KUKA KRL program: ps_a_lta_res_x01.src, ps_a_lta_res_x01.dat

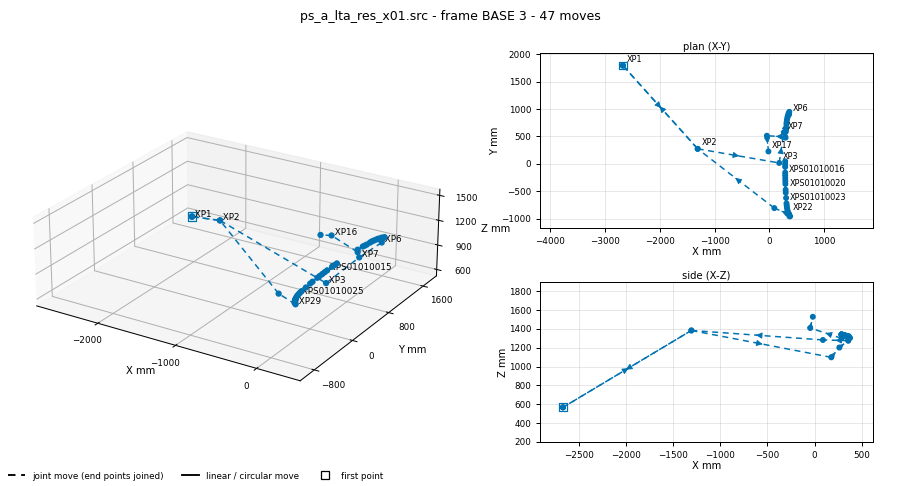
[picture p0: tool path of ps_a_lta_res_x01.src in frame BASE 3, 47 of 49 moves have a stored position in this frame; points joined in program order, loops and branches not executed]
--- ps_a_lta_res_x01.src ---
&ACCESS RVO1
&REL 2
&PARAM DISKPATH = Program/AXOR_ATEGO
DEF ps_a_lta_res_x01( )

;FOLD INI;%{PE}
  ;FOLD BASISTECH INI
    GLOBAL INTERRUPT DECL 3 WHEN $STOPMESS==TRUE DO IR_STOPM ( )
    INTERRUPT ON 3
    BAS (#INITMOV,0 )
  ;ENDFOLD (BASISTECH INI)
;FOLD SPOTTECH INI
USERSPOT(#INIT)
;ENDFOLD (SPOTTECH INI)
;FOLD GRIPPERTECH INI
USER_GRP(0,DUMMY,DUMMY,GDEFAULT)
;ENDFOLD (GRIPPERTECH INI)
  ;FOLD USER INI
    ;Make your modifications here

  ;ENDFOLD (USER INI)
;ENDFOLD (INI)

; Caracterizacao dos meios de producao
; Changes: Solda Respot - ATEGO LTA
; Versao Atual: 07/04/2016
; Ferramenta: GUN X1
; Name: P13.090-R6

chk_w4_wechs_ok ( )     ; CHECK GUN X1

if MaxStandMenge (4) then
  MaxStandmengeErreicht (4)
endif
if Elektrodenwechsel (4) then
 ; e_fraes4 ()
endif

;FOLD PTP P1 Vel=100 % PDAT1 Tool[4]:Gun X1 Base[3]:Atego/Axor;%{PE}%R 8.2.24,%MKUKATPBASIS,%CMOVE,%VPTP,%P 1:PTP, 2:P1, 3:, 5:100, 7:PDAT1
$BWDSTART=FALSE
PDAT_ACT=PPDAT1
FDAT_ACT=FP1
BAS(#PTP_PARAMS,100)
PTP XP1
;ENDFOLD

;FOLD ; Aguarda Liberacao p/ Soldar Respot;%{PE}%R8.3,%MKUKATPBASIS,%CCOMMENT,%VNORMAL,%P 2: Aguarda Liberacao p/ Soldar Respot
;ENDFOLD
;FOLD OUT 3346 'MAGAZINE 3 OCUPADO' State=TRUE ;%{PE}%R 8.2.24,%MKUKATPBASIS,%COUT,%VOUTX,%P 2:3346, 3:MAGAZINE 3 OCUPADO, 5:TRUE, 6:
$OUT[3346]=TRUE
;ENDFOLD
;FOLD WAIT FOR ( IN 3346 'LIB. ROBO SOLDAR RESPOT (ATEGO/AXOR)' );%{PE}%R 8.2.24,%MKUKATPBASIS,%CEXT_WAIT_FOR,%VEXT_WAIT_FOR,%P 2:, 4:, 5:$IN, 6:3346, 7:LIB. ROBO SOLDAR RESPOT (ATEGO/AXOR), 9:
WAIT FOR  ( $IN[3346] )
;ENDFOLD
;FOLD OUT 3346 'MAGAZINE 3 OCUPADO' State=FALSE ;%{PE}%R 8.2.24,%MKUKATPBASIS,%COUT,%VOUTX,%P 2:3346, 3:MAGAZINE 3 OCUPADO, 5:FALSE, 6:
$OUT[3346]=FALSE
;ENDFOLD

;FOLD ; Liga intertravamento  com R4;%{PE}%R8.3,%MKUKATPBASIS,%CCOMMENT,%VNORMAL,%P 2: Liga intertravamento  com R4
;ENDFOLD
;FOLD ; Intertravamento 15 do R4 equivalente ao Intertravamento 15 no R6;%{PE}%R 8.2.24,%MKUKATPBASIS,%CCOMMENT,%VNORMAL,%P 2:Intertravamento 15 do R4 equivalente ao Intertravamento 15 no R6
;ENDFOLD
;FOLD Collision.Monitoring_15_On ;%{PE}%MKUKATPUSER

COLLSTOP( 15, 1 ) ;not Interrupt-Controlled

;ENDFOLD

;FOLD PTP P2 CONT Vel=100 % PDAT2 Tool[4]:Gun X1 Base[3]:Atego/Axor;%{PE}%R 8.2.24,%MKUKATPBASIS,%CMOVE,%VPTP,%P 1:PTP, 2:P2, 3:C_PTP, 5:100, 7:PDAT2
$BWDSTART=FALSE
PDAT_ACT=PPDAT2
FDAT_ACT=FP2
BAS(#PTP_PARAMS,100)
PTP XP2 C_PTP
;ENDFOLD
;FOLD PTP P3 CONT Vel=100 % PDAT3 Tool[4]:Gun X1 Base[3]:Atego/Axor;%{PE}%R 8.2.24,%MKUKATPBASIS,%CMOVE,%VPTP,%P 1:PTP, 2:P3, 3:C_PTP, 5:100, 7:PDAT3
$BWDSTART=FALSE
PDAT_ACT=PPDAT3
FDAT_ACT=FP3
BAS(#PTP_PARAMS,100)
PTP XP3 C_PTP
;ENDFOLD
;FOLD PTP P7 CONT Vel=100 % PDAT6 Tool[4]:Gun X1 Base[3]:Atego/Axor;%{PE}%R 8.2.24,%MKUKATPBASIS,%CMOVE,%VPTP,%P 1:PTP, 2:P7, 3:C_PTP, 5:100, 7:PDAT6
$BWDSTART=FALSE
PDAT_ACT=PPDAT6
FDAT_ACT=FP7
BAS(#PTP_PARAMS,100)
PTP XP7 C_PTP
;ENDFOLD
;FOLD PTP P6 Vel=100 % PDAT5 Tool[4]:Gun X1 Base[3]:Atego/Axor;%{PE}%R 8.2.24,%MKUKATPBASIS,%CMOVE,%VPTP,%P 1:PTP, 2:P6, 3:, 5:100, 7:PDAT5
$BWDSTART=FALSE
PDAT_ACT=PPDAT5
FDAT_ACT=FP6
BAS(#PTP_PARAMS,100)
PTP XP6
;ENDFOLD

;FOLD ; SWP_60_9640;%{PE}%R8.3,%MKUKATPBASIS,%CCOMMENT,%VNORMAL,%P 2: SWP_60_9640
;ENDFOLD
;FOLD LIN PS01010002 CPDAT6 SPOT Gun=2 RETR CLS PgNo1=182 ACTIVE=1 Tool[4]:Gun X1 Base[3]:Atego/Axor;%{PE}%R 8.2.2,%MKUKATPSPOT,%CSPOT,%VLIN,%P 1:LIN, 2:PS01010002, 3:, 5:2, 7:CPDAT6, 10:2, 12:#FIRST, 14:#CLO, 16:182, 18:1, 20:0, 22:0, 24:1, 25:NORMAL
$BWDSTART=FALSE
LDAT_ACT=LCPDAT6
FDAT_ACT=FPS01010002
BAS(#CP_PARAMS,LCPDAT6.VEL)
S_ACT.GUN=2
S_ACT.PAIR=SDEFAULT.PAIR
S_ACT.RETR=#CLO
S_ACT.CLO_TM=1
S_ACT.PGNO1=182
S_ACT.PGNO2=SDEFAULT.PGNO2
S_ACT.PRESS1=SDEFAULT.PRESS1
S_ACT.PRESS2=SDEFAULT.PRESS2
S_READY=FALSE
LIN XPS01010002
USERSPOT(#SPOT, S_ACT)
WAIT FOR S_READY

;ENDFOLD
;FOLD LIN P9 Vel=2 m/s CPDAT5 Tool[4]:Gun X1 Base[3]:Atego/Axor;%{PE}%R 8.2.24,%MKUKATPBASIS,%CMOVE,%VLIN,%P 1:LIN, 2:P9, 3:, 5:2, 7:CPDAT5
$BWDSTART=FALSE
LDAT_ACT=LCPDAT5
FDAT_ACT=FP9
BAS(#CP_PARAMS,2)
LIN XP9
;ENDFOLD

;FOLD ; SWP_60_9638;%{PE}%R8.3,%MKUKATPBASIS,%CCOMMENT,%VNORMAL,%P 2: SWP_60_9638
;ENDFOLD
;FOLD LIN PS01010003 CPDAT4 SPOT Gun=2 RETR CLS PgNo1=182 ACTIVE=1 Tool[4]:Gun X1 Base[3]:Atego/Axor;%{PE}%R 8.2.2,%MKUKATPSPOT,%CSPOT,%VLIN,%P 1:LIN, 2:PS01010003, 3:, 5:2, 7:CPDAT4, 10:2, 12:#FIRST, 14:#CLO, 16:182, 18:1, 20:0, 22:0, 24:1, 25:NORMAL
$BWDSTART=FALSE
LDAT_ACT=LCPDAT4
FDAT_ACT=FPS01010003
BAS(#CP_PARAMS,LCPDAT4.VEL)
S_ACT.GUN=2
S_ACT.PAIR=SDEFAULT.PAIR
S_ACT.RETR=#CLO
S_ACT.CLO_TM=1
S_ACT.PGNO1=182
S_ACT.PGNO2=SDEFAULT.PGNO2
S_ACT.PRESS1=SDEFAULT.PRESS1
S_ACT.PRESS2=SDEFAULT.PRESS2
S_READY=FALSE
LIN XPS01010003
USERSPOT(#SPOT, S_ACT)
WAIT FOR S_READY

;ENDFOLD

;FOLD LIN P10 Vel=2 m/s CPDAT3 Tool[4]:Gun X1 Base[3]:Atego/Axor;%{PE}%R 8.2.24,%MKUKATPBASIS,%CMOVE,%VLIN,%P 1:LIN, 2:P10, 3:, 5:2, 7:CPDAT3
$BWDSTART=FALSE
LDAT_ACT=LCPDAT3
FDAT_ACT=FP10
BAS(#CP_PARAMS,2)
LIN XP10
;ENDFOLD

;FOLD ; SWP_60_9636;%{PE}%R8.3,%MKUKATPBASIS,%CCOMMENT,%VNORMAL,%P 2: SWP_60_9636
;ENDFOLD
;FOLD LIN PS01010004 CPDAT7 SPOT Gun=2 RETR CLS PgNo1=185 ACTIVE=1 Tool[4]:Gun X1 Base[3]:Atego/Axor;%{PE}%R 8.2.2,%MKUKATPSPOT,%CSPOT,%VLIN,%P 1:LIN, 2:PS01010004, 3:, 5:2, 7:CPDAT7, 10:2, 12:#FIRST, 14:#CLO, 16:185, 18:1, 20:0, 22:0, 24:1, 25:NORMAL
$BWDSTART=FALSE
LDAT_ACT=LCPDAT7
FDAT_ACT=FPS01010004
BAS(#CP_PARAMS,LCPDAT7.VEL)
S_ACT.GUN=2
S_ACT.PAIR=SDEFAULT.PAIR
S_ACT.RETR=#CLO
S_ACT.CLO_TM=1
S_ACT.PGNO1=185
S_ACT.PGNO2=SDEFAULT.PGNO2
S_ACT.PRESS1=SDEFAULT.PRESS1
S_ACT.PRESS2=SDEFAULT.PRESS2
S_READY=FALSE
LIN XPS01010004
USERSPOT(#SPOT, S_ACT)
WAIT FOR S_READY

;ENDFOLD

;FOLD ; SWP_60_9634;%{PE}%R8.3,%MKUKATPBASIS,%CCOMMENT,%VNORMAL,%P 2: SWP_60_9634
;ENDFOLD
;FOLD LIN PS01010005 CPDAT8 SPOT Gun=2 RETR CLS PgNo1=181 ACTIVE=1 Tool[4]:Gun X1 Base[3]:Atego/Axor;%{PE}%R 8.2.2,%MKUKATPSPOT,%CSPOT,%VLIN,%P 1:LIN, 2:PS01010005, 3:, 5:2, 7:CPDAT8, 10:2, 12:#FIRST, 14:#CLO, 16:181, 18:1, 20:0, 22:0, 24:1, 25:NORMAL
$BWDSTART=FALSE
LDAT_ACT=LCPDAT8
FDAT_ACT=FPS01010005
BAS(#CP_PARAMS,LCPDAT8.VEL)
S_ACT.GUN=2
S_ACT.PAIR=SDEFAULT.PAIR
S_ACT.RETR=#CLO
S_ACT.CLO_TM=1
S_ACT.PGNO1=181
S_ACT.PGNO2=SDEFAULT.PGNO2
S_ACT.PRESS1=SDEFAULT.PRESS1
S_ACT.PRESS2=SDEFAULT.PRESS2
S_READY=FALSE
LIN XPS01010005
USERSPOT(#SPOT, S_ACT)
WAIT FOR S_READY

;ENDFOLD

;FOLD ; SWP_60_9632;%{PE}%R8.3,%MKUKATPBASIS,%CCOMMENT,%VNORMAL,%P 2: SWP_60_9632
;ENDFOLD
;FOLD LIN PS01010006 CPDAT9 SPOT Gun=2 RETR CLS PgNo1=181 ACTIVE=1 Tool[4]:Gun X1 Base[3]:Atego/Axor;%{PE}%R 8.2.2,%MKUKATPSPOT,%CSPOT,%VLIN,%P 1:LIN, 2:PS01010006, 3:, 5:2, 7:CPDAT9, 10:2, 12:#FIRST, 14:#CLO, 16:181, 18:1, 20:0, 22:0, 24:1, 25:NORMAL
$BWDSTART=FALSE
LDAT_ACT=LCPDAT9
FDAT_ACT=FPS01010006
BAS(#CP_PARAMS,LCPDAT9.VEL)
S_ACT.GUN=2
S_ACT.PAIR=SDEFAULT.PAIR
S_ACT.RETR=#CLO
S_ACT.CLO_TM=1
S_ACT.PGNO1=181
S_ACT.PGNO2=SDEFAULT.PGNO2
S_ACT.PRESS1=SDEFAULT.PRESS1
S_ACT.PRESS2=SDEFAULT.PRESS2
S_READY=FALSE
LIN XPS01010006
USERSPOT(#SPOT, S_ACT)
WAIT FOR S_READY

;ENDFOLD

;FOLD ; SWP_60_9630;%{PE}%R8.3,%MKUKATPBASIS,%CCOMMENT,%VNORMAL,%P 2: SWP_60_9630
;ENDFOLD
;FOLD LIN PS01010008 CPDAT11 SPOT Gun=2 RETR CLS PgNo1=181 ACTIVE=1 Tool[4]:Gun X1 Base[3]:Atego/Axor;%{PE}%R 8.2.2,%MKUKATPSPOT,%CSPOT,%VLIN,%P 1:LIN, 2:PS01010008, 3:, 5:2, 7:CPDAT11, 10:2, 12:#FIRST, 14:#CLO, 16:181, 18:1, 20:0, 22:0, 24:1, 25:NORMAL
$BWDSTART=FALSE
LDAT_ACT=LCPDAT11
FDAT_ACT=FPS01010008
BAS(#CP_PARAMS,LCPDAT11.VEL)
S_ACT.GUN=2
S_ACT.PAIR=SDEFAULT.PAIR
S_ACT.RETR=#CLO
S_ACT.CLO_TM=1
S_ACT.PGNO1=181
S_ACT.PGNO2=SDEFAULT.PGNO2
S_ACT.PRESS1=SDEFAULT.PRESS1
S_ACT.PRESS2=SDEFAULT.PRESS2
S_READY=FALSE
LIN XPS01010008
USERSPOT(#SPOT, S_ACT)
WAIT FOR S_READY

;ENDFOLD

;FOLD ; SWP_60_9628;%{PE}%R8.3,%MKUKATPBASIS,%CCOMMENT,%VNORMAL,%P 2: SWP_60_9628
;ENDFOLD
;FOLD LIN PS01010009 CPDAT12 SPOT Gun=2 RETR CLS PgNo1=181 ACTIVE=1 Tool[4]:Gun X1 Base[3]:Atego/Axor;%{PE}%R 8.2.2,%MKUKATPSPOT,%CSPOT,%VLIN,%P 1:LIN, 2:PS01010009, 3:, 5:2, 7:CPDAT12, 10:2, 12:#FIRST, 14:#CLO, 16:181, 18:1, 20:0, 22:0, 24:1, 25:NORMAL
$BWDSTART=FALSE
LDAT_ACT=LCPDAT12
FDAT_ACT=FPS01010009
BAS(#CP_PARAMS,LCPDAT12.VEL)
S_ACT.GUN=2
S_ACT.PAIR=SDEFAULT.PAIR
S_ACT.RETR=#CLO
S_ACT.CLO_TM=1
S_ACT.PGNO1=181
S_ACT.PGNO2=SDEFAULT.PGNO2
S_ACT.PRESS1=SDEFAULT.PRESS1
S_ACT.PRESS2=SDEFAULT.PRESS2
S_READY=FALSE
LIN XPS01010009
USERSPOT(#SPOT, S_ACT)
WAIT FOR S_READY

;ENDFOLD

;FOLD LIN P13 CONT Vel=2 m/s CPDAT16 Tool[4]:Gun X1 Base[3]:Atego/Axor;%{PE}%R 8.2.24,%MKUKATPBASIS,%CMOVE,%VLIN,%P 1:LIN, 2:P13, 3:C_DIS, 5:2, 7:CPDAT16
$BWDSTART=FALSE
LDAT_ACT=LCPDAT16
FDAT_ACT=FP13
BAS(#CP_PARAMS,2)
LIN XP13 C_DIS
;ENDFOLD
;FOLD ; SWP_60_9624;%{PE}%R8.3,%MKUKATPBASIS,%CCOMMENT,%VNORMAL,%P 2: SWP_60_9624
;ENDFOLD
;FOLD LIN PS01010010 CPDAT15 SPOT Gun=2 RETR CLS PgNo1=186 ACTIVE=1 Tool[4]:Gun X1 Base[3]:Atego/Axor;%{PE}%R 8.2.2,%MKUKATPSPOT,%CSPOT,%VLIN,%P 1:LIN, 2:PS01010010, 3:, 5:2, 7:CPDAT15, 10:2, 12:#FIRST, 14:#CLO, 16:186, 18:1, 20:0, 22:0, 24:1, 25:NORMAL
$BWDSTART=FALSE
LDAT_ACT=LCPDAT15
FDAT_ACT=FPS01010010
BAS(#CP_PARAMS,LCPDAT15.VEL)
S_ACT.GUN=2
S_ACT.PAIR=SDEFAULT.PAIR
S_ACT.RETR=#CLO
S_ACT.CLO_TM=1
S_ACT.PGNO1=186
S_ACT.PGNO2=SDEFAULT.PGNO2
S_ACT.PRESS1=SDEFAULT.PRESS1
S_ACT.PRESS2=SDEFAULT.PRESS2
S_READY=FALSE
LIN XPS01010010
USERSPOT(#SPOT, S_ACT)
WAIT FOR S_READY

;ENDFOLD

;FOLD ; SWP_60_9622;%{PE}%R8.3,%MKUKATPBASIS,%CCOMMENT,%VNORMAL,%P 2: SWP_60_9622
;ENDFOLD
;FOLD LIN PS01010011 CPDAT17 SPOT Gun=2 RETR CLS PgNo1=181 ACTIVE=1 Tool[4]:Gun X1 Base[3]:Atego/Axor;%{PE}%R 8.2.2,%MKUKATPSPOT,%CSPOT,%VLIN,%P 1:LIN, 2:PS01010011, 3:, 5:2, 7:CPDAT17, 10:2, 12:#FIRST, 14:#CLO, 16:181, 18:1, 20:0, 22:0, 24:1, 25:NORMAL
$BWDSTART=FALSE
LDAT_ACT=LCPDAT17
FDAT_ACT=FPS01010011
BAS(#CP_PARAMS,LCPDAT17.VEL)
S_ACT.GUN=2
S_ACT.PAIR=SDEFAULT.PAIR
S_ACT.RETR=#CLO
S_ACT.CLO_TM=1
S_ACT.PGNO1=181
S_ACT.PGNO2=SDEFAULT.PGNO2
S_ACT.PRESS1=SDEFAULT.PRESS1
S_ACT.PRESS2=SDEFAULT.PRESS2
S_READY=FALSE
LIN XPS01010011
USERSPOT(#SPOT, S_ACT)
WAIT FOR S_READY

;ENDFOLD

;FOLD ; SWP_60_9618;%{PE}%R8.3,%MKUKATPBASIS,%CCOMMENT,%VNORMAL,%P 2: SWP_60_9618
;ENDFOLD
;FOLD LIN PS01010012 CPDAT18 SPOT Gun=2 RETR CLS PgNo1=181 ACTIVE=1 Tool[4]:Gun X1 Base[3]:Atego/Axor;%{PE}%R 8.2.2,%MKUKATPSPOT,%CSPOT,%VLIN,%P 1:LIN, 2:PS01010012, 3:, 5:2, 7:CPDAT18, 10:2, 12:#FIRST, 14:#CLO, 16:181, 18:1, 20:0, 22:0, 24:1, 25:NORMAL
$BWDSTART=FALSE
LDAT_ACT=LCPDAT18
FDAT_ACT=FPS01010012
BAS(#CP_PARAMS,LCPDAT18.VEL)
S_ACT.GUN=2
S_ACT.PAIR=SDEFAULT.PAIR
S_ACT.RETR=#CLO
S_ACT.CLO_TM=1
S_ACT.PGNO1=181
S_ACT.PGNO2=SDEFAULT.PGNO2
S_ACT.PRESS1=SDEFAULT.PRESS1
S_ACT.PRESS2=SDEFAULT.PRESS2
S_READY=FALSE
LIN XPS01010012
USERSPOT(#SPOT, S_ACT)
WAIT FOR S_READY

;ENDFOLD

;FOLD LIN P14 Vel=2 m/s CPDAT19 Tool[4]:Gun X1 Base[3]:Atego/Axor;%{PE}%R 8.2.24,%MKUKATPBASIS,%CMOVE,%VLIN,%P 1:LIN, 2:P14, 3:, 5:2, 7:CPDAT19
$BWDSTART=FALSE
LDAT_ACT=LCPDAT19
FDAT_ACT=FP14
BAS(#CP_PARAMS,2)
LIN XP14
;ENDFOLD
;FOLD PTP P16 Vel=100 % PDAT12 Tool[4]:Gun X1 Base[3]:Atego/Axor;%{PE}%R 8.2.24,%MKUKATPBASIS,%CMOVE,%VPTP,%P 1:PTP, 2:P16, 3:, 5:100, 7:PDAT12
$BWDSTART=FALSE
PDAT_ACT=PPDAT12
FDAT_ACT=FP16
BAS(#PTP_PARAMS,100)
PTP XP16
;ENDFOLD
;FOLD PTP P17 CONT Vel=100 % PDAT13 Tool[4]:Gun X1 Base[3]:Atego/Axor;%{PE}%R 8.2.24,%MKUKATPBASIS,%CMOVE,%VPTP,%P 1:PTP, 2:P17, 3:C_PTP, 5:100, 7:PDAT13
$BWDSTART=FALSE
PDAT_ACT=PPDAT13
FDAT_ACT=FP17
BAS(#PTP_PARAMS,100)
PTP XP17 C_PTP
;ENDFOLD
;FOLD PTP P19 CONT Vel=100 % PDAT14 Tool[5]:Gripper Geo G01 00 Base[0];%{PE}%R 8.2.24,%MKUKATPBASIS,%CMOVE,%VPTP,%P 1:PTP, 2:P19, 3:C_PTP, 5:100, 7:PDAT14
$BWDSTART=FALSE
PDAT_ACT=PPDAT14
FDAT_ACT=FP19
BAS(#PTP_PARAMS,100)
PTP XP19 C_PTP
;ENDFOLD
;FOLD PTP P20 Vel=100 % PDAT15 Tool[5]:Gripper Geo G01 00 Base[0];%{PE}%R 8.2.24,%MKUKATPBASIS,%CMOVE,%VPTP,%P 1:PTP, 2:P20, 3:, 5:100, 7:PDAT15
$BWDSTART=FALSE
PDAT_ACT=PPDAT15
FDAT_ACT=FP20
BAS(#PTP_PARAMS,100)
PTP XP20
;ENDFOLD

;FOLD ; SWP_60_9602;%{PE}%R8.3,%MKUKATPBASIS,%CCOMMENT,%VNORMAL,%P 2: SWP_60_9602
;ENDFOLD
;FOLD LIN PS01010013 CPDAT20 SPOT Gun=2 RETR CLS PgNo1=181 ACTIVE=1 Tool[4]:Gun X1 Base[3]:Atego/Axor;%{PE}%R 8.2.2,%MKUKATPSPOT,%CSPOT,%VLIN,%P 1:LIN, 2:PS01010013, 3:, 5:2, 7:CPDAT20, 10:2, 12:#FIRST, 14:#CLO, 16:181, 18:1, 20:0, 22:0, 24:1, 25:NORMAL
$BWDSTART=FALSE
LDAT_ACT=LCPDAT20
FDAT_ACT=FPS01010013
BAS(#CP_PARAMS,LCPDAT20.VEL)
S_ACT.GUN=2
S_ACT.PAIR=SDEFAULT.PAIR
S_ACT.RETR=#CLO
S_ACT.CLO_TM=1
S_ACT.PGNO1=181
S_ACT.PGNO2=SDEFAULT.PGNO2
S_ACT.PRESS1=SDEFAULT.PRESS1
S_ACT.PRESS2=SDEFAULT.PRESS2
S_READY=FALSE
LIN XPS01010013
USERSPOT(#SPOT, S_ACT)
WAIT FOR S_READY

;ENDFOLD

;FOLD ; SWP_60_9600;%{PE}%R8.3,%MKUKATPBASIS,%CCOMMENT,%VNORMAL,%P 2: SWP_60_9600
;ENDFOLD
;FOLD LIN PS01010007 CPDAT10 SPOT Gun=2 RETR CLS PgNo1=186 ACTIVE=1 Tool[4]:Gun X1 Base[3]:Atego/Axor;%{PE}%R 8.2.2,%MKUKATPSPOT,%CSPOT,%VLIN,%P 1:LIN, 2:PS01010007, 3:, 5:2, 7:CPDAT10, 10:2, 12:#FIRST, 14:#CLO, 16:186, 18:1, 20:0, 22:0, 24:1, 25:NORMAL
$BWDSTART=FALSE
LDAT_ACT=LCPDAT10
FDAT_ACT=FPS01010007
BAS(#CP_PARAMS,LCPDAT10.VEL)
S_ACT.GUN=2
S_ACT.PAIR=SDEFAULT.PAIR
S_ACT.RETR=#CLO
S_ACT.CLO_TM=1
S_ACT.PGNO1=186
S_ACT.PGNO2=SDEFAULT.PGNO2
S_ACT.PRESS1=SDEFAULT.PRESS1
S_ACT.PRESS2=SDEFAULT.PRESS2
S_READY=FALSE
LIN XPS01010007
USERSPOT(#SPOT, S_ACT)
WAIT FOR S_READY

;ENDFOLD

;FOLD ; SWP_60_9601;%{PE}%R8.3,%MKUKATPBASIS,%CCOMMENT,%VNORMAL,%P 2: SWP_60_9601
;ENDFOLD
;FOLD LIN PS01010014 CPDAT21 SPOT Gun=2 RETR CLS PgNo1=181 ACTIVE=1 Tool[4]:Gun X1 Base[3]:Atego/Axor;%{PE}%R 8.2.2,%MKUKATPSPOT,%CSPOT,%VLIN,%P 1:LIN, 2:PS01010014, 3:, 5:2, 7:CPDAT21, 10:2, 12:#FIRST, 14:#CLO, 16:181, 18:1, 20:0, 22:0, 24:1, 25:NORMAL
$BWDSTART=FALSE
LDAT_ACT=LCPDAT21
FDAT_ACT=FPS01010014
BAS(#CP_PARAMS,LCPDAT21.VEL)
S_ACT.GUN=2
S_ACT.PAIR=SDEFAULT.PAIR
S_ACT.RETR=#CLO
S_ACT.CLO_TM=1
S_ACT.PGNO1=181
S_ACT.PGNO2=SDEFAULT.PGNO2
S_ACT.PRESS1=SDEFAULT.PRESS1
S_ACT.PRESS2=SDEFAULT.PRESS2
S_READY=FALSE
LIN XPS01010014
USERSPOT(#SPOT, S_ACT)
WAIT FOR S_READY

;ENDFOLD

;FOLD ; SWP_60_9605;%{PE}%R8.3,%MKUKATPBASIS,%CCOMMENT,%VNORMAL,%P 2: SWP_60_9605
;ENDFOLD
;FOLD LIN PS01010015 CPDAT22 SPOT Gun=2 RETR CLS PgNo1=181 ACTIVE=1 Tool[4]:Gun X1 Base[3]:Atego/Axor;%{PE}%R 8.2.2,%MKUKATPSPOT,%CSPOT,%VLIN,%P 1:LIN, 2:PS01010015, 3:, 5:2, 7:CPDAT22, 10:2, 12:#FIRST, 14:#CLO, 16:181, 18:1, 20:0, 22:0, 24:1, 25:NORMAL
$BWDSTART=FALSE
LDAT_ACT=LCPDAT22
FDAT_ACT=FPS01010015
BAS(#CP_PARAMS,LCPDAT22.VEL)
S_ACT.GUN=2
S_ACT.PAIR=SDEFAULT.PAIR
S_ACT.RETR=#CLO
S_ACT.CLO_TM=1
S_ACT.PGNO1=181
S_ACT.PGNO2=SDEFAULT.PGNO2
S_ACT.PRESS1=SDEFAULT.PRESS1
S_ACT.PRESS2=SDEFAULT.PRESS2
S_READY=FALSE
LIN XPS01010015
USERSPOT(#SPOT, S_ACT)
WAIT FOR S_READY

;ENDFOLD

;FOLD ; SWP_60_9607;%{PE}%R8.3,%MKUKATPBASIS,%CCOMMENT,%VNORMAL,%P 2: SWP_60_9607
;ENDFOLD
;FOLD LIN PS01010016 CPDAT23 SPOT Gun=2 RETR CLS PgNo1=181 ACTIVE=1 Tool[4]:Gun X1 Base[3]:Atego/Axor;%{PE}%R 8.2.2,%MKUKATPSPOT,%CSPOT,%VLIN,%P 1:LIN, 2:PS01010016, 3:, 5:2, 7:CPDAT23, 10:2, 12:#FIRST, 14:#CLO, 16:181, 18:1, 20:0, 22:0, 24:1, 25:NORMAL
$BWDSTART=FALSE
LDAT_ACT=LCPDAT23
FDAT_ACT=FPS01010016
BAS(#CP_PARAMS,LCPDAT23.VEL)
S_ACT.GUN=2
S_ACT.PAIR=SDEFAULT.PAIR
S_ACT.RETR=#CLO
S_ACT.CLO_TM=1
S_ACT.PGNO1=181
S_ACT.PGNO2=SDEFAULT.PGNO2
S_ACT.PRESS1=SDEFAULT.PRESS1
S_ACT.PRESS2=SDEFAULT.PRESS2
S_READY=FALSE
LIN XPS01010016
USERSPOT(#SPOT, S_ACT)
WAIT FOR S_READY

;ENDFOLD

;FOLD ; SWP_60_9609;%{PE}%R8.3,%MKUKATPBASIS,%CCOMMENT,%VNORMAL,%P 2: SWP_60_9609
;ENDFOLD
;FOLD LIN PS01010017 CPDAT24 SPOT Gun=2 RETR CLS PgNo1=181 ACTIVE=1 Tool[4]:Gun X1 Base[3]:Atego/Axor;%{PE}%R 8.2.2,%MKUKATPSPOT,%CSPOT,%VLIN,%P 1:LIN, 2:PS01010017, 3:, 5:2, 7:CPDAT24, 10:2, 12:#FIRST, 14:#CLO, 16:181, 18:1, 20:0, 22:0, 24:1, 25:NORMAL
$BWDSTART=FALSE
LDAT_ACT=LCPDAT24
FDAT_ACT=FPS01010017
BAS(#CP_PARAMS,LCPDAT24.VEL)
S_ACT.GUN=2
S_ACT.PAIR=SDEFAULT.PAIR
S_ACT.RETR=#CLO
S_ACT.CLO_TM=1
S_ACT.PGNO1=181
S_ACT.PGNO2=SDEFAULT.PGNO2
S_ACT.PRESS1=SDEFAULT.PRESS1
S_ACT.PRESS2=SDEFAULT.PRESS2
S_READY=FALSE
LIN XPS01010017
USERSPOT(#SPOT, S_ACT)
WAIT FOR S_READY

;ENDFOLD

;FOLD ; SWP_60_9611;%{PE}%R8.3,%MKUKATPBASIS,%CCOMMENT,%VNORMAL,%P 2: SWP_60_9611
;ENDFOLD
;FOLD LIN PS01010018 CPDAT25 SPOT Gun=2 RETR CLS PgNo1=181 ACTIVE=1 Tool[4]:Gun X1 Base[3]:Atego/Axor;%{PE}%R 8.2.2,%MKUKATPSPOT,%CSPOT,%VLIN,%P 1:LIN, 2:PS01010018, 3:, 5:2, 7:CPDAT25, 10:2, 12:#FIRST, 14:#CLO, 16:181, 18:1, 20:0, 22:0, 24:1, 25:NORMAL
$BWDSTART=FALSE
LDAT_ACT=LCPDAT25
FDAT_ACT=FPS01010018
BAS(#CP_PARAMS,LCPDAT25.VEL)
S_ACT.GUN=2
S_ACT.PAIR=SDEFAULT.PAIR
S_ACT.RETR=#CLO
S_ACT.CLO_TM=1
S_ACT.PGNO1=181
S_ACT.PGNO2=SDEFAULT.PGNO2
S_ACT.PRESS1=SDEFAULT.PRESS1
S_ACT.PRESS2=SDEFAULT.PRESS2
S_READY=FALSE
LIN XPS01010018
USERSPOT(#SPOT, S_ACT)
WAIT FOR S_READY

;ENDFOLD

;FOLD ; SWP_60_9613;%{PE}%R8.3,%MKUKATPBASIS,%CCOMMENT,%VNORMAL,%P 2: SWP_60_9613
;ENDFOLD
;FOLD LIN PS01010019 CPDAT26 SPOT Gun=2 RETR CLS PgNo1=181 ACTIVE=1 Tool[4]:Gun X1 Base[3]:Atego/Axor;%{PE}%R 8.2.2,%MKUKATPSPOT,%CSPOT,%VLIN,%P 1:LIN, 2:PS01010019, 3:, 5:2, 7:CPDAT26, 10:2, 12:#FIRST, 14:#CLO, 16:181, 18:1, 20:0, 22:0, 24:1, 25:NORMAL
$BWDSTART=FALSE
LDAT_ACT=LCPDAT26
FDAT_ACT=FPS01010019
BAS(#CP_PARAMS,LCPDAT26.VEL)
S_ACT.GUN=2
S_ACT.PAIR=SDEFAULT.PAIR
S_ACT.RETR=#CLO
S_ACT.CLO_TM=1
S_ACT.PGNO1=181
S_ACT.PGNO2=SDEFAULT.PGNO2
S_ACT.PRESS1=SDEFAULT.PRESS1
S_ACT.PRESS2=SDEFAULT.PRESS2
S_READY=FALSE
LIN XPS01010019
USERSPOT(#SPOT, S_ACT)
WAIT FOR S_READY

;ENDFOLD

;FOLD ; SWP_60_9617;%{PE}%R8.3,%MKUKATPBASIS,%CCOMMENT,%VNORMAL,%P 2: SWP_60_9617
;ENDFOLD
;FOLD LIN PS01010020 CPDAT27 SPOT Gun=2 RETR CLS PgNo1=181 ACTIVE=1 Tool[4]:Gun X1 Base[3]:Atego/Axor;%{PE}%R 8.2.2,%MKUKATPSPOT,%CSPOT,%VLIN,%P 1:LIN, 2:PS01010020, 3:, 5:2, 7:CPDAT27, 10:2, 12:#FIRST, 14:#CLO, 16:181, 18:1, 20:0, 22:0, 24:1, 25:NORMAL
$BWDSTART=FALSE
LDAT_ACT=LCPDAT27
FDAT_ACT=FPS01010020
BAS(#CP_PARAMS,LCPDAT27.VEL)
S_ACT.GUN=2
S_ACT.PAIR=SDEFAULT.PAIR
S_ACT.RETR=#CLO
S_ACT.CLO_TM=1
S_ACT.PGNO1=181
S_ACT.PGNO2=SDEFAULT.PGNO2
S_ACT.PRESS1=SDEFAULT.PRESS1
S_ACT.PRESS2=SDEFAULT.PRESS2
S_READY=FALSE
LIN XPS01010020
USERSPOT(#SPOT, S_ACT)
WAIT FOR S_READY

;ENDFOLD

;FOLD ; SWP_60_9619;%{PE}%R8.3,%MKUKATPBASIS,%CCOMMENT,%VNORMAL,%P 2: SWP_60_9619
;ENDFOLD
;FOLD LIN PS01010021 CPDAT28 SPOT Gun=2 RETR CLS PgNo1=181 ACTIVE=1 Tool[4]:Gun X1 Base[3]:Atego/Axor;%{PE}%R 8.2.2,%MKUKATPSPOT,%CSPOT,%VLIN,%P 1:LIN, 2:PS01010021, 3:, 5:2, 7:CPDAT28, 10:2, 12:#FIRST, 14:#CLO, 16:181, 18:1, 20:0, 22:0, 24:1, 25:NORMAL
$BWDSTART=FALSE
LDAT_ACT=LCPDAT28
FDAT_ACT=FPS01010021
BAS(#CP_PARAMS,LCPDAT28.VEL)
S_ACT.GUN=2
S_ACT.PAIR=SDEFAULT.PAIR
S_ACT.RETR=#CLO
S_ACT.CLO_TM=1
S_ACT.PGNO1=181
S_ACT.PGNO2=SDEFAULT.PGNO2
S_ACT.PRESS1=SDEFAULT.PRESS1
S_ACT.PRESS2=SDEFAULT.PRESS2
S_READY=FALSE
LIN XPS01010021
USERSPOT(#SPOT, S_ACT)
WAIT FOR S_READY

;ENDFOLD

;FOLD ; SWP_60_9623;%{PE}%R8.3,%MKUKATPBASIS,%CCOMMENT,%VNORMAL,%P 2: SWP_60_9623
;ENDFOLD
;FOLD LIN PS01010022 CPDAT29 SPOT Gun=2 RETR CLS PgNo1=186 ACTIVE=1 Tool[4]:Gun X1 Base[3]:Atego/Axor;%{PE}%R 8.2.2,%MKUKATPSPOT,%CSPOT,%VLIN,%P 1:LIN, 2:PS01010022, 3:, 5:2, 7:CPDAT29, 10:2, 12:#FIRST, 14:#CLO, 16:186, 18:1, 20:0, 22:0, 24:1, 25:NORMAL
$BWDSTART=FALSE
LDAT_ACT=LCPDAT29
FDAT_ACT=FPS01010022
BAS(#CP_PARAMS,LCPDAT29.VEL)
S_ACT.GUN=2
S_ACT.PAIR=SDEFAULT.PAIR
S_ACT.RETR=#CLO
S_ACT.CLO_TM=1
S_ACT.PGNO1=186
S_ACT.PGNO2=SDEFAULT.PGNO2
S_ACT.PRESS1=SDEFAULT.PRESS1
S_ACT.PRESS2=SDEFAULT.PRESS2
S_READY=FALSE
LIN XPS01010022
USERSPOT(#SPOT, S_ACT)
WAIT FOR S_READY

;ENDFOLD

;FOLD ; SWP_60_9627(old 9625);%{PE}%R8.3,%MKUKATPBASIS,%CCOMMENT,%VNORMAL,%P 2: SWP_60_9627(old 9625)
;ENDFOLD
;FOLD LIN PS01010023 CPDAT30 SPOT Gun=2 RETR CLS PgNo1=186 ACTIVE=1 Tool[4]:Gun X1 Base[3]:Atego/Axor;%{PE}%R 8.2.2,%MKUKATPSPOT,%CSPOT,%VLIN,%P 1:LIN, 2:PS01010023, 3:, 5:2, 7:CPDAT30, 10:2, 12:#FIRST, 14:#CLO, 16:186, 18:1, 20:0, 22:0, 24:1, 25:NORMAL
$BWDSTART=FALSE
LDAT_ACT=LCPDAT30
FDAT_ACT=FPS01010023
BAS(#CP_PARAMS,LCPDAT30.VEL)
S_ACT.GUN=2
S_ACT.PAIR=SDEFAULT.PAIR
S_ACT.RETR=#CLO
S_ACT.CLO_TM=1
S_ACT.PGNO1=186
S_ACT.PGNO2=SDEFAULT.PGNO2
S_ACT.PRESS1=SDEFAULT.PRESS1
S_ACT.PRESS2=SDEFAULT.PRESS2
S_READY=FALSE
LIN XPS01010023
USERSPOT(#SPOT, S_ACT)
WAIT FOR S_READY

;ENDFOLD

;FOLD ; Desliga intertravamento  com R4;%{PE}%R8.3,%MKUKATPBASIS,%CCOMMENT,%VNORMAL,%P 2: Desliga intertravamento  com R4
;ENDFOLD
;FOLD ; Intertravamento 15 do R4 equivalente ao Intertravamento 15 no R6;%{PE}%R 8.2.24,%MKUKATPBASIS,%CCOMMENT,%VNORMAL,%P 2:Intertravamento 15 do R4 equivalente ao Intertravamento 15 no R6
;ENDFOLD
;FOLD Collision.Monitoring_15_Off . ;%{PE}%MKUKATPUSER

COLLSTOP( 15, 2+0 )

;ENDFOLD

;FOLD ; SWP_60_9629;%{PE}%R8.3,%MKUKATPBASIS,%CCOMMENT,%VNORMAL,%P 2: SWP_60_9629
;ENDFOLD
;FOLD LIN PS01010024 CPDAT31 SPOT Gun=2 RETR CLS PgNo1=181 ACTIVE=1 Tool[4]:Gun X1 Base[3]:Atego/Axor;%{PE}%R 8.2.2,%MKUKATPSPOT,%CSPOT,%VLIN,%P 1:LIN, 2:PS01010024, 3:, 5:2, 7:CPDAT31, 10:2, 12:#FIRST, 14:#CLO, 16:181, 18:1, 20:0, 22:0, 24:1, 25:NORMAL
$BWDSTART=FALSE
LDAT_ACT=LCPDAT31
FDAT_ACT=FPS01010024
BAS(#CP_PARAMS,LCPDAT31.VEL)
S_ACT.GUN=2
S_ACT.PAIR=SDEFAULT.PAIR
S_ACT.RETR=#CLO
S_ACT.CLO_TM=1
S_ACT.PGNO1=181
S_ACT.PGNO2=SDEFAULT.PGNO2
S_ACT.PRESS1=SDEFAULT.PRESS1
S_ACT.PRESS2=SDEFAULT.PRESS2
S_READY=FALSE
LIN XPS01010024
USERSPOT(#SPOT, S_ACT)
WAIT FOR S_READY

;ENDFOLD

;FOLD ; SWP_60_9631;%{PE}%R8.3,%MKUKATPBASIS,%CCOMMENT,%VNORMAL,%P 2: SWP_60_9631
;ENDFOLD
;FOLD LIN PS01010025 CPDAT32 SPOT Gun=2 RETR CLS PgNo1=181 ACTIVE=1 Tool[4]:Gun X1 Base[3]:Atego/Axor;%{PE}%R 8.2.2,%MKUKATPSPOT,%CSPOT,%VLIN,%P 1:LIN, 2:PS01010025, 3:, 5:2, 7:CPDAT32, 10:2, 12:#FIRST, 14:#CLO, 16:181, 18:1, 20:0, 22:0, 24:1, 25:NORMAL
$BWDSTART=FALSE
LDAT_ACT=LCPDAT32
FDAT_ACT=FPS01010025
BAS(#CP_PARAMS,LCPDAT32.VEL)
S_ACT.GUN=2
S_ACT.PAIR=SDEFAULT.PAIR
S_ACT.RETR=#CLO
S_ACT.CLO_TM=1
S_ACT.PGNO1=181
S_ACT.PGNO2=SDEFAULT.PGNO2
S_ACT.PRESS1=SDEFAULT.PRESS1
S_ACT.PRESS2=SDEFAULT.PRESS2
S_READY=FALSE
LIN XPS01010025
USERSPOT(#SPOT, S_ACT)
WAIT FOR S_READY

;ENDFOLD

;FOLD ; SWP_60_9633;%{PE}%R8.3,%MKUKATPBASIS,%CCOMMENT,%VNORMAL,%P 2: SWP_60_9633
;ENDFOLD
;FOLD LIN PS01010026 CPDAT33 SPOT Gun=2 RETR CLS PgNo1=181 ACTIVE=1 Tool[4]:Gun X1 Base[3]:Atego/Axor;%{PE}%R 8.2.2,%MKUKATPSPOT,%CSPOT,%VLIN,%P 1:LIN, 2:PS01010026, 3:, 5:2, 7:CPDAT33, 10:2, 12:#FIRST, 14:#CLO, 16:181, 18:1, 20:0, 22:0, 24:1, 25:NORMAL
$BWDSTART=FALSE
LDAT_ACT=LCPDAT33
FDAT_ACT=FPS01010026
BAS(#CP_PARAMS,LCPDAT33.VEL)
S_ACT.GUN=2
S_ACT.PAIR=SDEFAULT.PAIR
S_ACT.RETR=#CLO
S_ACT.CLO_TM=1
S_ACT.PGNO1=181
S_ACT.PGNO2=SDEFAULT.PGNO2
S_ACT.PRESS1=SDEFAULT.PRESS1
S_ACT.PRESS2=SDEFAULT.PRESS2
S_READY=FALSE
LIN XPS01010026
USERSPOT(#SPOT, S_ACT)
WAIT FOR S_READY

;ENDFOLD

;FOLD ; SWP_60_9635;%{PE}%R8.3,%MKUKATPBASIS,%CCOMMENT,%VNORMAL,%P 2: SWP_60_9635
;ENDFOLD
;FOLD LIN PS01010027 CPDAT34 SPOT Gun=2 RETR CLS PgNo1=185 ACTIVE=1 Tool[4]:Gun X1 Base[3]:Atego/Axor;%{PE}%R 8.2.2,%MKUKATPSPOT,%CSPOT,%VLIN,%P 1:LIN, 2:PS01010027, 3:, 5:2, 7:CPDAT34, 10:2, 12:#FIRST, 14:#CLO, 16:185, 18:1, 20:0, 22:0, 24:1, 25:NORMAL
$BWDSTART=FALSE
LDAT_ACT=LCPDAT34
FDAT_ACT=FPS01010027
BAS(#CP_PARAMS,LCPDAT34.VEL)
S_ACT.GUN=2
S_ACT.PAIR=SDEFAULT.PAIR
S_ACT.RETR=#CLO
S_ACT.CLO_TM=1
S_ACT.PGNO1=185
S_ACT.PGNO2=SDEFAULT.PGNO2
S_ACT.PRESS1=SDEFAULT.PRESS1
S_ACT.PRESS2=SDEFAULT.PRESS2
S_READY=FALSE
LIN XPS01010027
USERSPOT(#SPOT, S_ACT)
WAIT FOR S_READY

;ENDFOLD

;FOLD LIN P22 Vel=2 m/s CPDAT35 Tool[4]:Gun X1 Base[3]:Atego/Axor;%{PE}%R 8.2.24,%MKUKATPBASIS,%CMOVE,%VLIN,%P 1:LIN, 2:P22, 3:, 5:2, 7:CPDAT35
$BWDSTART=FALSE
LDAT_ACT=LCPDAT35
FDAT_ACT=FP22
BAS(#CP_PARAMS,2)
LIN XP22
;ENDFOLD

;FOLD ; SWP_60_9637;%{PE}%R8.3,%MKUKATPBASIS,%CCOMMENT,%VNORMAL,%P 2: SWP_60_9637
;ENDFOLD
;FOLD LIN PS01010028 CPDAT36 SPOT Gun=2 RETR CLS PgNo1=184 ACTIVE=1 Tool[4]:Gun X1 Base[3]:Atego/Axor;%{PE}%R 8.2.2,%MKUKATPSPOT,%CSPOT,%VLIN,%P 1:LIN, 2:PS01010028, 3:, 5:2, 7:CPDAT36, 10:2, 12:#FIRST, 14:#CLO, 16:184, 18:1, 20:0, 22:0, 24:1, 25:NORMAL
$BWDSTART=FALSE
LDAT_ACT=LCPDAT36
FDAT_ACT=FPS01010028
BAS(#CP_PARAMS,LCPDAT36.VEL)
S_ACT.GUN=2
S_ACT.PAIR=SDEFAULT.PAIR
S_ACT.RETR=#CLO
S_ACT.CLO_TM=1
S_ACT.PGNO1=184
S_ACT.PGNO2=SDEFAULT.PGNO2
S_ACT.PRESS1=SDEFAULT.PRESS1
S_ACT.PRESS2=SDEFAULT.PRESS2
S_READY=FALSE
LIN XPS01010028
USERSPOT(#SPOT, S_ACT)
WAIT FOR S_READY

;ENDFOLD

;FOLD LIN P23 Vel=2 m/s CPDAT37 Tool[4]:Gun X1 Base[3]:Atego/Axor;%{PE}%R 8.2.24,%MKUKATPBASIS,%CMOVE,%VLIN,%P 1:LIN, 2:P23, 3:, 5:2, 7:CPDAT37
$BWDSTART=FALSE
LDAT_ACT=LCPDAT37
FDAT_ACT=FP23
BAS(#CP_PARAMS,2)
LIN XP23
;ENDFOLD
;FOLD LIN P24 Vel=2 m/s CPDAT38 Tool[4]:Gun X1 Base[3]:Atego/Axor;%{PE}%R 8.2.24,%MKUKATPBASIS,%CMOVE,%VLIN,%P 1:LIN, 2:P24, 3:, 5:2, 7:CPDAT38
$BWDSTART=FALSE
LDAT_ACT=LCPDAT38
FDAT_ACT=FP24
BAS(#CP_PARAMS,2)
LIN XP24
;ENDFOLD

;FOLD ; Liga intertravamento  com R4;%{PE}%R8.3,%MKUKATPBASIS,%CCOMMENT,%VNORMAL,%P 2: Liga intertravamento  com R4
;ENDFOLD
;FOLD ; Intertravamento 15 do R4 equivalente ao Intertravamento 15 no R6;%{PE}%R 8.2.24,%MKUKATPBASIS,%CCOMMENT,%VNORMAL,%P 2:Intertravamento 15 do R4 equivalente ao Intertravamento 15 no R6
;ENDFOLD
;FOLD Collision.Monitoring_15_On ;%{PE}%MKUKATPUSER

COLLSTOP( 15, 1 ) ;not Interrupt-Controlled

;ENDFOLD

;FOLD ; SWP_60_9639;%{PE}%R8.3,%MKUKATPBASIS,%CCOMMENT,%VNORMAL,%P 2: SWP_60_9639
;ENDFOLD
;FOLD LIN PS01010029 CPDAT40 SPOT Gun=2 RETR OPN PgNo1=184 ACTIVE=1 Tool[4]:Gun X1 Base[3]:Atego/Axor;%{PE}%R 8.2.2,%MKUKATPSPOT,%CSPOT,%VLIN,%P 1:LIN, 2:PS01010029, 3:, 5:2, 7:CPDAT40, 10:2, 12:#FIRST, 14:#OPN, 16:184, 18:1, 20:0, 22:0, 24:1, 25:NORMAL
$BWDSTART=FALSE
LDAT_ACT=LCPDAT40
FDAT_ACT=FPS01010029
BAS(#CP_PARAMS,LCPDAT40.VEL)
S_ACT.GUN=2
S_ACT.PAIR=SDEFAULT.PAIR
S_ACT.RETR=#OPN
S_ACT.CLO_TM=1
S_ACT.PGNO1=184
S_ACT.PGNO2=SDEFAULT.PGNO2
S_ACT.PRESS1=SDEFAULT.PRESS1
S_ACT.PRESS2=SDEFAULT.PRESS2
S_READY=FALSE
LIN XPS01010029
USERSPOT(#SPOT, S_ACT)
WAIT FOR S_READY

;ENDFOLD

;FOLD LIN P29 Vel=2 m/s CPDAT41 Tool[4]:Gun X1 Base[3]:Atego/Axor;%{PE}%R 8.2.24,%MKUKATPBASIS,%CMOVE,%VLIN,%P 1:LIN, 2:P29, 3:, 5:2, 7:CPDAT41
$BWDSTART=FALSE
LDAT_ACT=LCPDAT41
FDAT_ACT=FP29
BAS(#CP_PARAMS,2)
LIN XP29
;ENDFOLD
;FOLD PTP P30 CONT Vel=100 % PDAT19 Tool[4]:Gun X1 Base[3]:Atego/Axor;%{PE}%R 8.2.24,%MKUKATPBASIS,%CMOVE,%VPTP,%P 1:PTP, 2:P30, 3:C_PTP, 5:100, 7:PDAT19
$BWDSTART=FALSE
PDAT_ACT=PPDAT19
FDAT_ACT=FP30
BAS(#PTP_PARAMS,100)
PTP XP30 C_PTP
;ENDFOLD
;FOLD PTP P31 CONT Vel=100 % PDAT20 Tool[4]:Gun X1 Base[3]:Atego/Axor;%{PE}%R 8.2.24,%MKUKATPBASIS,%CMOVE,%VPTP,%P 1:PTP, 2:P31, 3:C_PTP, 5:100, 7:PDAT20
$BWDSTART=FALSE
PDAT_ACT=PPDAT20
FDAT_ACT=FP31
BAS(#PTP_PARAMS,100)
PTP XP31 C_PTP
;ENDFOLD
;FOLD PTP P32 Vel=100 % PDAT21 Tool[4]:Gun X1 Base[3]:Atego/Axor;%{PE}%R 8.2.24,%MKUKATPBASIS,%CMOVE,%VPTP,%P 1:PTP, 2:P32, 3:, 5:100, 7:PDAT21
$BWDSTART=FALSE
PDAT_ACT=PPDAT21
FDAT_ACT=FP32
BAS(#PTP_PARAMS,100)
PTP XP32
;ENDFOLD

;FOLD ; Desliga intertravamento  com R4;%{PE}%R8.3,%MKUKATPBASIS,%CCOMMENT,%VNORMAL,%P 2: Desliga intertravamento  com R4
;ENDFOLD
;FOLD ; Intertravamento 15 do R4 equivalente ao Intertravamento 15 no R6;%{PE}%R 8.2.24,%MKUKATPBASIS,%CCOMMENT,%VNORMAL,%P 2:Intertravamento 15 do R4 equivalente ao Intertravamento 15 no R6
;ENDFOLD
;FOLD Collision.Monitoring_15_Off . ;%{PE}%MKUKATPUSER

COLLSTOP( 15, 2+0 )

;ENDFOLD

;FOLD ; Libera Dispositivo;%{PE}%R8.3,%MKUKATPBASIS,%CCOMMENT,%VNORMAL,%P 2: Libera Dispositivo
;ENDFOLD
;FOLD OUT 3346 'MAGAZINE 3 OCUPADO' State=TRUE CONT;%{PE}%R 8.2.24,%MKUKATPBASIS,%COUT,%VOUTX,%P 2:3346, 3:MAGAZINE 3 OCUPADO, 5:TRUE, 6:CONTINUE
CONTINUE
$OUT[3346]=TRUE
;ENDFOLD

if FraesAnf (4) then
f_fraes4 ()
endif

;FOLD PTP P33 Vel=100 % PDAT22 Tool[4]:Gun X1 Base[3]:Atego/Axor;%{PE}%R 8.2.24,%MKUKATPBASIS,%CMOVE,%VPTP,%P 1:PTP, 2:P33, 3:, 5:100, 7:PDAT22
$BWDSTART=FALSE
PDAT_ACT=PPDAT22
FDAT_ACT=FP33
BAS(#PTP_PARAMS,100)
PTP XP33
;ENDFOLD
END

--- ps_a_lta_res_x01.dat ---
&ACCESS RVO1
&REL 2
&PARAM DISKPATH = Program/AXOR_ATEGO
DEFDAT ps_a_lta_res_x01
;FOLD EXTERNAL DECLARATIONS;%{PE}%MKUKATPBASIS,%CEXT,%VCOMMON,%P
;FOLD BASISTECH EXT;%{PE}%MKUKATPBASIS,%CEXT,%VEXT,%P
EXT  BAS (BAS_COMMAND  :IN,REAL  :IN )
DECL INT SUCCESS
;ENDFOLD (BASISTECH EXT)
;FOLD USER EXT;%{E}%MKUKATPUSER,%CEXT,%VEXT,%P
;Make your modifications here
;ENDFOLD (USER EXT)
;ENDFOLD (EXTERNAL DECLARATIONS)

;# ============ START PATH : ps_a_lta_res_x01 =============
DECL FDAT Fxp8={TOOL_NO 4,BASE_NO 3,IPO_FRAME #BASE,POINT2[] " "}
DECL PDAT PP_OLP1={VEL 100.0,ACC 100.0,APO_DIST 0.0}
DECL E6POS Xxp8={X -2671.84912,Y 1793.97302,Z 566.737,A -2.42820001,B 58.0560989,C 1.01139998,S 2,T 3}
DECL FDAT Fxp10={TOOL_NO 4,BASE_NO 3,IPO_FRAME #BASE,POINT2[] " "}
DECL PDAT PP_OLP2={VEL 100.0,ACC 100.0,APO_DIST 0.0}
DECL E6POS Xxp10={X -1308.078,Y 274.528015,Z 1383.49097,A -11.6739998,B 10.1196003,C -74.1667023,S 2,T 11}
DECL FDAT Fxp20={TOOL_NO 4,BASE_NO 3,IPO_FRAME #BASE,POINT2[] " "}
DECL PDAT PP_OLP3={VEL 100.0,ACC 50.0,APO_DIST 0.0}
DECL E6POS Xxp20={X 178.113007,Y 17.2910004,Z 1098.07605,A 11.9650002,B 9.40390015,C -82.9534988,S 2,T 11}
DECL FDAT Fx1005={TOOL_NO 4,BASE_NO 3,IPO_FRAME #BASE,POINT2[] " "}
DECL E6POS Xx1005={X 338.674988,Y 935.075989,Z 1286.09204,A 34.7946014,B -38.0540009,C -65.3376999,S 2,T 11}
DECL LDAT LL_OLP1={VEL 2.0,ACC 100.0,APO_DIST 1.0,APO_FAC 0.0,ORI_TYP #VAR,CIRC_TYP #BASE,JERK_FAC 50.0}
DECL FDAT Fx1010={TOOL_NO 4,BASE_NO 3,IPO_FRAME #BASE,POINT2[] " "}
DECL E6POS Xx1010={X 371.002014,Y 957.528015,Z 1316.90698,A 34.7947006,B -38.0540009,C -65.3376007,S 2,T 11}
DECL LDAT LL_OLP2={VEL 2.0,ACC 100.0,APO_DIST 1.0,APO_FAC 0.0,ORI_TYP #VAR,CIRC_TYP #BASE,JERK_FAC 50.0}
DECL FDAT Fxswp_6={TOOL_NO 4,BASE_NO 3,IPO_FRAME #BASE,POINT2[] " "}
DECL SPOT_TYPE SS_OLP1={GUN 2,PAIR #FIRST,RETR #CLO,CLO_TM 1,PGNO1 182,PRESS1 0.0,PGNO2 0,PRESS2 0.0}
DECL E6POS Xxswp_6={X 361.389008,Y 946.713989,Z 1327.31006,A 34.7943993,B -38.0540009,C -65.3374023,S 2,T 11}
DECL LDAT LL_OLP3={VEL 2.0,ACC 100.0,APO_DIST 0.0,APO_FAC 0.0,ORI_TYP #VAR,CIRC_TYP #BASE,JERK_FAC 50.0}
DECL FDAT Fx1015={TOOL_NO 4,BASE_NO 3,IPO_FRAME #BASE,POINT2[] " "}
DECL E6POS Xx1015={X 371.001007,Y 957.525024,Z 1316.90601,A 34.7947006,B -38.0540009,C -65.3376999,S 2,T 11}
DECL LDAT LL_OLP4={VEL 2.0,ACC 100.0,APO_DIST 1.0,APO_FAC 0.0,ORI_TYP #VAR,CIRC_TYP #BASE,JERK_FAC 50.0}
DECL FDAT Fxswp_6_1={TOOL_NO 4,BASE_NO 3,IPO_FRAME #BASE,POINT2[] " "}
DECL SPOT_TYPE SS_OLP2={GUN 2,PAIR #FIRST,RETR #CLO,CLO_TM 1,PGNO1 182,PRESS1 0.0,PGNO2 0,PRESS2 0.0}
DECL E6POS Xxswp_6_1={X 344.567993,Y 912.476013,Z 1332.31006,A 51.0245018,B -39.1311989,C -64.2306976,S 2,T 11}
DECL LDAT LL_OLP5={VEL 2.0,ACC 100.0,APO_DIST 0.0,APO_FAC 0.0,ORI_TYP #VAR,CIRC_TYP #BASE,JERK_FAC 50.0}
DECL FDAT Fx1030={TOOL_NO 4,BASE_NO 3,IPO_FRAME #BASE,POINT2[] " "}
DECL E6POS Xx1030={X 344.359985,Y 891.754028,Z 1333.81995,A 56.9338989,B -41.1417999,C -62.901001,S 2,T 11}
DECL LDAT LL_OLP6={VEL 2.0,ACC 100.0,APO_DIST 1.0,APO_FAC 0.0,ORI_TYP #VAR,CIRC_TYP #BASE,JERK_FAC 50.0}
DECL FDAT Fxswp_6_2={TOOL_NO 4,BASE_NO 3,IPO_FRAME #BASE,POINT2[] " "}
DECL SPOT_TYPE SS_OLP3={GUN 2,PAIR #FIRST,RETR #CLO,CLO_TM 1,PGNO1 185,PRESS1 0.0,PGNO2 0,PRESS2 0.0}
DECL E6POS Xxswp_6_2={X 331.682007,Y 863.525024,Z 1333.83398,A 56.9338989,B -41.1417999,C -62.901001,S 2,T 11}
DECL LDAT LL_OLP7={VEL 2.0,ACC 100.0,APO_DIST 0.0,APO_FAC 0.0,ORI_TYP #VAR,CIRC_TYP #BASE,JERK_FAC 50.0}
DECL FDAT Fxswp_6_3={TOOL_NO 4,BASE_NO 3,IPO_FRAME #BASE,POINT2[] " "}
DECL SPOT_TYPE SS_OLP4={GUN 2,PAIR #FIRST,RETR #CLO,CLO_TM 1,PGNO1 181,PRESS1 0.0,PGNO2 0,PRESS2 0.0}
DECL E6POS Xxswp_6_3={X 324.64801,Y 835.888977,Z 1335.92297,A 64.0038986,B -37.8157997,C -65.0102997,S 2,T 11}
DECL LDAT LL_OLP8={VEL 2.0,ACC 100.0,APO_DIST 0.0,APO_FAC 0.0,ORI_TYP #VAR,CIRC_TYP #BASE,JERK_FAC 50.0}
DECL FDAT Fxswp_6_4={TOOL_NO 4,BASE_NO 3,IPO_FRAME #BASE,POINT2[] " "}
DECL SPOT_TYPE SS_OLP5={GUN 2,PAIR #FIRST,RETR #CLO,CLO_TM 1,PGNO1 181,PRESS1 0.0,PGNO2 0,PRESS2 0.0}
DECL E6POS Xxswp_6_4={X 318.389008,Y 798.062012,Z 1336.797,A 63.0040016,B -41.4422989,C -63.5331001,S 2,T 11}
DECL LDAT LL_OLP9={VEL 2.0,ACC 100.0,APO_DIST 0.0,APO_FAC 0.0,ORI_TYP #VAR,CIRC_TYP #BASE,JERK_FAC 50.0}
DECL FDAT Fxswp_6_5={TOOL_NO 4,BASE_NO 3,IPO_FRAME #BASE,POINT2[] " "}
DECL SPOT_TYPE SS_OLP6={GUN 2,PAIR #FIRST,RETR #CLO,CLO_TM 1,PGNO1 181,PRESS1 0.0,PGNO2 0,PRESS2 0.0}
DECL E6POS Xxswp_6_5={X 313.28299,Y 758.213989,Z 1338.11304,A 65.8960037,B -39.6694984,C -64.0615997,S 2,T 11}
DECL LDAT LL_OLP10={VEL 2.0,ACC 100.0,APO_DIST 0.0,APO_FAC 0.0,ORI_TYP #VAR,CIRC_TYP #BASE,JERK_FAC 50.0}
DECL FDAT Fxswp_6_6={TOOL_NO 4,BASE_NO 3,IPO_FRAME #BASE,POINT2[] " "}
DECL SPOT_TYPE SS_OLP7={GUN 2,PAIR #FIRST,RETR #CLO,CLO_TM 1,PGNO1 181,PRESS1 0.0,PGNO2 0,PRESS2 0.0}
DECL E6POS Xxswp_6_6={X 309.087006,Y 718.695007,Z 1339.03503,A 69.3459015,B -38.6236992,C -68.3812027,S 2,T 11}
DECL LDAT LL_OLP11={VEL 2.0,ACC 100.0,APO_DIST 0.0,APO_FAC 0.0,ORI_TYP #VAR,CIRC_TYP #BASE,JERK_FAC 50.0}
DECL FDAT Fx1035={TOOL_NO 4,BASE_NO 3,IPO_FRAME #BASE,POINT2[] " "}
DECL E6POS Xx1035={X 297.544006,Y 716.080017,Z 1298.703,A 69.3459015,B -38.6237984,C -68.3811035,S 2,T 11}
DECL LDAT LL_OLP12={VEL 2.0,ACC 100.0,APO_DIST 1.0,APO_FAC 0.0,ORI_TYP #VAR,CIRC_TYP #BASE,JERK_FAC 50.0}
DECL FDAT Fx1040={TOOL_NO 4,BASE_NO 3,IPO_FRAME #BASE,POINT2[] " "}
DECL PDAT PP_OLP4={VEL 100.0,ACC 100.0,APO_DIST 0.0}
DECL E6POS Xx1040={X 290.720001,Y 611.52002,Z 1294.58899,A 70.504303,B -35.8750992,C -65.2176971,S 2,T 11}
DECL FDAT Fxswp_6_7={TOOL_NO 4,BASE_NO 3,IPO_FRAME #BASE,POINT2[] " "}
DECL SPOT_TYPE SS_OLP8={GUN 2,PAIR #FIRST,RETR #CLO,CLO_TM 1,PGNO1 186,PRESS1 0.0,PGNO2 0,PRESS2 0.0}
DECL E6POS Xxswp_6_7={X 302.175995,Y 615.903992,Z 1338.88904,A 70.504097,B -35.8751984,C -65.2176971,S 2,T 11}
DECL LDAT LL_OLP13={VEL 2.0,ACC 100.0,APO_DIST 0.0,APO_FAC 0.0,ORI_TYP #VAR,CIRC_TYP #BASE,JERK_FAC 50.0}
DECL FDAT Fxswp_6_8={TOOL_NO 4,BASE_NO 3,IPO_FRAME #BASE,POINT2[] " "}
DECL SPOT_TYPE SS_OLP9={GUN 2,PAIR #FIRST,RETR #CLO,CLO_TM 1,PGNO1 181,PRESS1 0.0,PGNO2 0,PRESS2 0.0}
DECL E6POS Xxswp_6_8={X 298.696991,Y 582.974976,Z 1340.22302,A 71.1110001,B -36.0985985,C -65.1601028,S 2,T 11}
DECL LDAT LL_OLP14={VEL 2.0,ACC 100.0,APO_DIST 0.0,APO_FAC 0.0,ORI_TYP #VAR,CIRC_TYP #BASE,JERK_FAC 50.0}
DECL FDAT Fxswp_6_9={TOOL_NO 4,BASE_NO 3,IPO_FRAME #BASE,POINT2[] " "}
DECL SPOT_TYPE SS_OLP10={GUN 2,PAIR #FIRST,RETR #CLO,CLO_TM 1,PGNO1 181,PRESS1 0.0,PGNO2 0,PRESS2 0.0}
DECL E6POS Xxswp_6_9={X 293.197998,Y 476.902008,Z 1341.17297,A 67.3917007,B -43.7565002,C -61.9462013,S 2,T 11}
DECL LDAT LL_OLP15={VEL 2.0,ACC 100.0,APO_DIST 0.0,APO_FAC 0.0,ORI_TYP #VAR,CIRC_TYP #BASE,JERK_FAC 50.0}
DECL FDAT Fxl1045={TOOL_NO 4,BASE_NO 3,IPO_FRAME #BASE,POINT2[] " "}
DECL E6POS Xxl045={X 283.067993,Y 502.061005,Z 1308.948,A 69.0100021,B -41.4696007,C -63.0419998,S 2,T 11}
DECL LDAT LL_OLP16={VEL 2.0,ACC 100.0,APO_DIST 1.0,APO_FAC 0.0,ORI_TYP #VAR,CIRC_TYP #BASE,JERK_FAC 50.0}
DECL FDAT Fx1050={TOOL_NO 4,BASE_NO 3,IPO_FRAME #BASE,POINT2[] " "}
DECL PDAT PP_OLP5={VEL 100.0,ACC 100.0,APO_DIST 0.0}
DECL E6POS Xx1050={X -45.6539993,Y 513.651978,Z 1409.17297,A 70.8384018,B -38.6459007,C -64.219101,S 2,T 11}
DECL FDAT Fx1055={TOOL_NO 4,BASE_NO 3,IPO_FRAME #BASE,POINT2[] " "}
DECL PDAT PP_OLP6={VEL 100.0,ACC 100.0,APO_DIST 0.0}
DECL E6POS Xx1055={X -18.0699997,Y 226.630005,Z 1528.59204,A -52.2551003,B -66.299202,C 40.457901,S 2,T 11}
DECL FDAT Fx1060={TOOL_NO 4,BASE_NO 3,IPO_FRAME #BASE,POINT2[] " "}
DECL PDAT PP_OLP7={VEL 100.0,ACC 100.0,APO_DIST 0.0}
DECL E6POS Xxl060={X -83.6139984,Y 28.8789997,Z 1405.45605,A -82.8872986,B -20.2294998,C 69.417099,S 2,T 11}
DECL FDAT Fx1065={TOOL_NO 4,BASE_NO 3,IPO_FRAME #BASE,POINT2[] " "}
DECL PDAT PP_OLP8={VEL 100.0,ACC 100.0,APO_DIST 0.0}
DECL E6POS Xx1065={X 286.222992,Y 27.2730007,Z 1301.41101,A -82.8872986,B -20.2294998,C 69.417099,S 2,T 11}
DECL FDAT Fxswp_6_10={TOOL_NO 4,BASE_NO 3,IPO_FRAME #BASE,POINT2[] " "}
DECL SPOT_TYPE SS_OLP11={GUN 2,PAIR #FIRST,RETR #CLO,CLO_TM 1,PGNO1 181,PRESS1 0.0,PGNO2 0,PRESS2 0.0}
DECL E6POS Xxswp_6_10={X 287.351013,Y 48.5550003,Z 1346.63,A -82.1261978,B -22.1051006,C 69.1417999,S 2,T 11}
DECL LDAT LL_OLP17={VEL 2.0,ACC 100.0,APO_DIST 0.0,APO_FAC 0.0,ORI_TYP #VAR,CIRC_TYP #BASE,JERK_FAC 50.0}
DECL FDAT Fxswp_6_11={TOOL_NO 4,BASE_NO 3,IPO_FRAME #BASE,POINT2[] " "}
DECL SPOT_TYPE SS_OLP12={GUN 2,PAIR #FIRST,RETR #CLO,CLO_TM 1,PGNO1 186,PRESS1 0.0,PGNO2 0,PRESS2 0.0}
DECL E6POS Xxswp_6_11={X 287.300995,Y -3.58200002,Z 1345.09399,A -81.5048981,B -23.1126995,C 68.9759979,S 2,T 11}
DECL LDAT LL_OLP18={VEL 2.0,ACC 100.0,APO_DIST 0.0,APO_FAC 0.0,ORI_TYP #VAR,CIRC_TYP #BASE,JERK_FAC 50.0}
DECL FDAT Fxswp_6_12={TOOL_NO 4,BASE_NO 3,IPO_FRAME #BASE,POINT2[] " "}
DECL SPOT_TYPE SS_OLP13={GUN 2,PAIR #FIRST,RETR #CLO,CLO_TM 1,PGNO1 181,PRESS1 0.0,PGNO2 0,PRESS2 0.0}
DECL E6POS Xxswp_6_12={X 285.257996,Y -52.1780014,Z 1346.73706,A -81.077301,B -23.4216995,C 68.9110031,S 2,T 11}
DECL LDAT LL_OLP19={VEL 2.0,ACC 100.0,APO_DIST 0.0,APO_FAC 0.0,ORI_TYP #VAR,CIRC_TYP #BASE,JERK_FAC 50.0}
DECL FDAT Fxswp_6_13={TOOL_NO 4,BASE_NO 3,IPO_FRAME #BASE,POINT2[] " "}
DECL SPOT_TYPE SS_OLP14={GUN 2,PAIR #FIRST,RETR #CLO,CLO_TM 1,PGNO1 181,PRESS1 0.0,PGNO2 0,PRESS2 0.0}
DECL E6POS Xxswp_6_13={X 286.690002,Y -156.309998,Z 1346.33704,A -81.3834,B -21.8426991,C 69.1763992,S 2,T 11}
DECL LDAT LL_OLP20={VEL 2.0,ACC 100.0,APO_DIST 0.0,APO_FAC 0.0,ORI_TYP #VAR,CIRC_TYP #BASE,JERK_FAC 50.0}
DECL FDAT Fxswp_6_14={TOOL_NO 4,BASE_NO 3,IPO_FRAME #BASE,POINT2[] " "}
DECL SPOT_TYPE SS_OLP15={GUN 2,PAIR #FIRST,RETR #CLO,CLO_TM 1,PGNO1 181,PRESS1 0.0,PGNO2 0,PRESS2 0.0}
DECL E6POS Xxswp_6_14={X 288.113007,Y -207.438004,Z 1345.89294,A -81.4317017,B -21.0953999,C 69.4869003,S 2,T 11}
DECL LDAT LL_OLP21={VEL 2.0,ACC 100.0,APO_DIST 0.0,APO_FAC 0.0,ORI_TYP #VAR,CIRC_TYP #BASE,JERK_FAC 50.0}
DECL FDAT Fxswp_6_15={TOOL_NO 4,BASE_NO 3,IPO_FRAME #BASE,POINT2[] " "}
DECL SPOT_TYPE SS_OLP16={GUN 2,PAIR #FIRST,RETR #CLO,CLO_TM 1,PGNO1 181,PRESS1 0.0,PGNO2 0,PRESS2 0.0}
DECL E6POS Xxswp_6_15={X 288.074005,Y -261.427002,Z 1345.67896,A -80.2265015,B -22.9715996,C 69.1436005,S 2,T 11}
DECL LDAT LL_OLP22={VEL 2.0,ACC 100.0,APO_DIST 0.0,APO_FAC 0.0,ORI_TYP #VAR,CIRC_TYP #BASE,JERK_FAC 50.0}
DECL FDAT Fxswp_6_16={TOOL_NO 4,BASE_NO 3,IPO_FRAME #BASE,POINT2[] " "}
DECL SPOT_TYPE SS_OLP17={GUN 2,PAIR #FIRST,RETR #CLO,CLO_TM 1,PGNO1 181,PRESS1 0.0,PGNO2 0,PRESS2 0.0}
DECL E6POS Xxswp_6_16={X 289.654999,Y -314.811005,Z 1344.66199,A -80.330101,B -22.3747005,C 69.0469971,S 2,T 11}
DECL LDAT LL_OLP23={VEL 2.0,ACC 100.0,APO_DIST 0.0,APO_FAC 0.0,ORI_TYP #VAR,CIRC_TYP #BASE,JERK_FAC 50.0}
DECL FDAT Fxswp_6_17={TOOL_NO 4,BASE_NO 3,IPO_FRAME #BASE,POINT2[] " "}
DECL SPOT_TYPE SS_OLP18={GUN 2,PAIR #FIRST,RETR #CLO,CLO_TM 1,PGNO1 181,PRESS1 0.0,PGNO2 0,PRESS2 0.0}
DECL E6POS Xxswp_6_17={X 290.39801,Y -367.192993,Z 1343.63098,A -80.1075974,B -22.1487007,C 69.3021011,S 2,T 11}
DECL LDAT LL_OLP24={VEL 2.0,ACC 100.0,APO_DIST 0.0,APO_FAC 0.0,ORI_TYP #VAR,CIRC_TYP #BASE,JERK_FAC 50.0}
DECL FDAT Fxswp_6_18={TOOL_NO 4,BASE_NO 3,IPO_FRAME #BASE,POINT2[] " "}
DECL SPOT_TYPE SS_OLP19={GUN 2,PAIR #FIRST,RETR #CLO,CLO_TM 1,PGNO1 181,PRESS1 0.0,PGNO2 0,PRESS2 0.0}
DECL E6POS Xxswp_6_18={X 293.604004,Y -472.330994,Z 1343.151,A -79.1949997,B -22.2735996,C 68.9171982,S 2,T 11}
DECL LDAT LL_OLP25={VEL 2.0,ACC 100.0,APO_DIST 0.0,APO_FAC 0.0,ORI_TYP #VAR,CIRC_TYP #BASE,JERK_FAC 50.0}
DECL FDAT Fxswp_6_19={TOOL_NO 4,BASE_NO 3,IPO_FRAME #BASE,POINT2[] " "}
DECL SPOT_TYPE SS_OLP20={GUN 2,PAIR #FIRST,RETR #CLO,CLO_TM 1,PGNO1 181,PRESS1 0.0,PGNO2 0,PRESS2 0.0}
DECL E6POS Xxswp_6_19={X 297.158997,Y -524.651001,Z 1342.01794,A -79.5855026,B -20.0948009,C 69.1838989,S 2,T 11}
DECL LDAT LL_OLP26={VEL 2.0,ACC 100.0,APO_DIST 0.0,APO_FAC 0.0,ORI_TYP #VAR,CIRC_TYP #BASE,JERK_FAC 50.0}
DECL FDAT Fxswp_6_20={TOOL_NO 4,BASE_NO 3,IPO_FRAME #BASE,POINT2[] " "}
DECL SPOT_TYPE SS_OLP21={GUN 2,PAIR #FIRST,RETR #CLO,CLO_TM 1,PGNO1 186,PRESS1 0.0,PGNO2 0,PRESS2 0.0}
DECL E6POS Xxswp_6_20={X 303.765015,Y -620.15802,Z 1339.09302,A -78.1246033,B -20.2479,C 69.1043015,S 2,T 11}
DECL LDAT LL_OLP27={VEL 2.0,ACC 100.0,APO_DIST 0.0,APO_FAC 0.0,ORI_TYP #VAR,CIRC_TYP #BASE,JERK_FAC 50.0}
DECL FDAT Fxswp_6_21={TOOL_NO 4,BASE_NO 3,IPO_FRAME #BASE,POINT2[] " "}
DECL SPOT_TYPE SS_OLP22={GUN 2,PAIR #FIRST,RETR #CLO,CLO_TM 1,PGNO1 186,PRESS1 0.0,PGNO2 0,PRESS2 0.0}
DECL E6POS Xxswp_6_21={X 310.752014,Y -721.088013,Z 1338.60901,A -76.822998,B -20.4850998,C 68.993103,S 2,T 11}
DECL LDAT LL_OLP28={VEL 2.0,ACC 100.0,APO_DIST 0.0,APO_FAC 0.0,ORI_TYP #VAR,CIRC_TYP #BASE,JERK_FAC 50.0}
DECL FDAT Fxswp_6_22={TOOL_NO 4,BASE_NO 3,IPO_FRAME #BASE,POINT2[] " "}
DECL SPOT_TYPE SS_OLP23={GUN 2,PAIR #FIRST,RETR #CLO,CLO_TM 1,PGNO1 181,PRESS1 0.0,PGNO2 0,PRESS2 0.0}
DECL E6POS Xxswp_6_22={X 315.821991,Y -759.333984,Z 1338.26697,A -76.5533981,B -18.2450008,C 69.2284012,S 2,T 11}
DECL LDAT LL_OLP29={VEL 2.0,ACC 100.0,APO_DIST 0.0,APO_FAC 0.0,ORI_TYP #VAR,CIRC_TYP #BASE,JERK_FAC 50.0}
DECL FDAT Fxswp_6_23={TOOL_NO 4,BASE_NO 3,IPO_FRAME #BASE,POINT2[] " "}
DECL SPOT_TYPE SS_OLP24={GUN 2,PAIR #FIRST,RETR #CLO,CLO_TM 1,PGNO1 181,PRESS1 0.0,PGNO2 0,PRESS2 0.0}
DECL E6POS Xxswp_6_23={X 322.985992,Y -795.739014,Z 1336.43103,A -74.3142014,B -18.2257996,C 69.5625992,S 2,T 11}
DECL LDAT LL_OLP30={VEL 2.0,ACC 100.0,APO_DIST 0.0,APO_FAC 0.0,ORI_TYP #VAR,CIRC_TYP #BASE,JERK_FAC 50.0}
DECL FDAT Fxswp_6_24={TOOL_NO 4,BASE_NO 3,IPO_FRAME #BASE,POINT2[] " "}
DECL SPOT_TYPE SS_OLP25={GUN 2,PAIR #FIRST,RETR #CLO,CLO_TM 1,PGNO1 181,PRESS1 0.0,PGNO2 0,PRESS2 0.0}
DECL E6POS Xxswp_6_24={X 324.492004,Y -834.676025,Z 1335.93298,A -72.3386002,B -19.9249992,C 69.1243973,S 2,T 11}
DECL LDAT LL_OLP31={VEL 2.0,ACC 100.0,APO_DIST 0.0,APO_FAC 0.0,ORI_TYP #VAR,CIRC_TYP #BASE,JERK_FAC 50.0}
DECL FDAT Fxswp_6_25={TOOL_NO 4,BASE_NO 3,IPO_FRAME #BASE,POINT2[] " "}
DECL SPOT_TYPE SS_OLP26={GUN 2,PAIR #FIRST,RETR #CLO,CLO_TM 1,PGNO1 185,PRESS1 0.0,PGNO2 0,PRESS2 0.0}
DECL E6POS Xxswp_6_25={X 332.988007,Y -867.458984,Z 1334.82397,A -72.338501,B -19.9249992,C 69.1243973,S 2,T 11}
DECL LDAT LL_OLP32={VEL 2.0,ACC 100.0,APO_DIST 0.0,APO_FAC 0.0,ORI_TYP #VAR,CIRC_TYP #BASE,JERK_FAC 50.0}
DECL FDAT Fx1075={TOOL_NO 4,BASE_NO 3,IPO_FRAME #BASE,POINT2[] " "}
DECL E6POS Xx1075={X 346.785004,Y -908.474976,Z 1323.55603,A -60.6660004,B -19.5358009,C 69.0325012,S 2,T 11}
DECL LDAT LL_OLP33={VEL 2.0,ACC 100.0,APO_DIST 0.0,APO_FAC 0.0,ORI_TYP #VAR,CIRC_TYP #BASE,JERK_FAC 50.0}
DECL FDAT Fxswp_6_26={TOOL_NO 4,BASE_NO 3,IPO_FRAME #BASE,POINT2[] " "}
DECL SPOT_TYPE SS_OLP27={GUN 2,PAIR #FIRST,RETR #CLO,CLO_TM 1,PGNO1 184,PRESS1 0.0,PGNO2 0,PRESS2 0.0}
DECL E6POS Xxswp_6_26={X 345.006012,Y -910.223999,Z 1329.95801,A -60.6665993,B -19.5352993,C 69.0325012,S 2,T 11}
DECL LDAT LL_OLP34={VEL 2.0,ACC 100.0,APO_DIST 0.0,APO_FAC 0.0,ORI_TYP #VAR,CIRC_TYP #BASE,JERK_FAC 50.0}
DECL FDAT Fx1080={TOOL_NO 4,BASE_NO 3,IPO_FRAME #BASE,POINT2[] " "}
DECL E6POS Xx1080={X 346.787994,Y -908.473022,Z 1323.55298,A -60.6660004,B -19.5358009,C 69.0325012,S 2,T 11}
DECL LDAT LL_OLP35={VEL 2.0,ACC 100.0,APO_DIST 0.0,APO_FAC 0.0,ORI_TYP #VAR,CIRC_TYP #BASE,JERK_FAC 50.0}
DECL FDAT Fx1085={TOOL_NO 4,BASE_NO 3,IPO_FRAME #BASE,POINT2[] " "}
DECL E6POS Xx1085={X 294.372986,Y -872.359009,Z 1225.72498,A -62.4161987,B -15.1138,C 69.5541992,S 2,T 11}
DECL LDAT LL_OLP36={VEL 2.0,ACC 100.0,APO_DIST 0.0,APO_FAC 0.0,ORI_TYP #VAR,CIRC_TYP #BASE,JERK_FAC 50.0}
DECL FDAT Fxl090={TOOL_NO 4,BASE_NO 3,IPO_FRAME #BASE,POINT2[] " "}
DECL PDAT PP_OLP9={VEL 100.0,ACC 100.0,APO_DIST 0.0}
DECL E6POS Xxl090={X 32.5680008,Y -978.309021,Z 1326.90503,A -56.223999,B -12.7813997,C 68.0599976,S 2,T 11}
DECL FDAT Fxl095={TOOL_NO 4,BASE_NO 3,IPO_FRAME #BASE,POINT2[] " "}
DECL PDAT PP_OLP10={VEL 100.0,ACC 100.0,APO_DIST 0.0}
DECL E6POS Xx1095={X 13.783,Y -909.382019,Z 1346.41699,A -50.0074005,B 9.56999969,C -160.030502,S 2,T 43}
DECL FDAT Fx1100={TOOL_NO 4,BASE_NO 3,IPO_FRAME #BASE,POINT2[] " "}
DECL E6POS Xxl100={X 342.721985,Y -966.474976,Z 1268.21399,A -47.9878006,B -7.45359993,C -109.351799,S 2,T 43}
DECL LDAT LL_OLP37={VEL 2.0,ACC 100.0,APO_DIST 0.0,APO_FAC 0.0,ORI_TYP #VAR,CIRC_TYP #BASE,JERK_FAC 50.0}
DECL FDAT Fx1105={TOOL_NO 4,BASE_NO 3,IPO_FRAME #BASE,POINT2[] " "}
DECL E6POS X1l105={X 363.707001,Y -963.538025,Z 1323.08704,A -47.9878006,B -7.45359993,C -109.351799,S 2,T 43}
DECL LDAT LL_OLP38={VEL 2.0,ACC 100.0,APO_DIST 0.0,APO_FAC 0.0,ORI_TYP #VAR,CIRC_TYP #BASE,JERK_FAC 50.0}
DECL FDAT Fxswp_6_27={TOOL_NO 4,BASE_NO 3,IPO_FRAME #BASE,POINT2[] " "}
DECL SPOT_TYPE SS_OLP28={GUN 2,PAIR #FIRST,RETR #CLO,CLO_TM 1,PGNO1 184,PRESS1 0.0,PGNO2 0,PRESS2 0.0}
DECL E6POS Xxswp_6_27={X 369.730988,Y -954.963013,Z 1322.66394,A -47.9878006,B -7.45349979,C -109.351898,S 2,T 43}
DECL LDAT LL_OLP39={VEL 2.0,ACC 100.0,APO_DIST 0.0,APO_FAC 0.0,ORI_TYP #VAR,CIRC_TYP #BASE,JERK_FAC 50.0}
DECL FDAT Fx1110={TOOL_NO 4,BASE_NO 3,IPO_FRAME #BASE,POINT2[] " "}
DECL E6POS Xx1110={X 363.707001,Y -963.531006,Z 1320.20398,A -47.9877014,B -7.45359993,C -109.351799,S 2,T 43}
DECL LDAT LL_OLP40={VEL 2.0,ACC 100.0,APO_DIST 0.0,APO_FAC 0.0,ORI_TYP #VAR,CIRC_TYP #BASE,JERK_FAC 50.0}
DECL FDAT Fx1115={TOOL_NO 4,BASE_NO 3,IPO_FRAME #BASE,POINT2[] " "}
DECL E6POS Xx1115={X 342.721985,Y -966.474976,Z 1268.21399,A -47.9878006,B -7.45359993,C -109.351799,S 2,T 43}
DECL LDAT LL_OLP41={VEL 2.0,ACC 100.0,APO_DIST 0.0,APO_FAC 0.0,ORI_TYP #VAR,CIRC_TYP #BASE,JERK_FAC 50.0}
DECL FDAT Fx1120={TOOL_NO 4,BASE_NO 3,IPO_FRAME #BASE,POINT2[] " "}
DECL PDAT PP_OLP11={VEL 100.0,ACC 100.0,APO_DIST 0.0}
DECL E6POS Xx1120={X 85.0699997,Y -691.823975,Z 1231.81799,A -47.9878006,B -7.45359993,C -109.351799,S 2,T 43}
DECL FDAT Fxp13={TOOL_NO 4,BASE_NO 3,IPO_FRAME #BASE,POINT2[] " "}
DECL PDAT PP_OLP12={VEL 100.0,ACC 50.0,APO_DIST 0.0}
DECL E6POS Xxp13={X 178.112,Y 17.2870007,Z 1098.07495,A 11.9647999,B 9.40400028,C -82.9534988,S 2,T 43}
DECL FDAT Fxp11={TOOL_NO 4,BASE_NO 3,IPO_FRAME #BASE,POINT2[] " "}
DECL PDAT PP_OLP13={VEL 100.0,ACC 100.0,APO_DIST 0.0}
DECL E6POS Xxp11={X -1308.07703,Y 274.528015,Z 1383.48901,A -11.6739998,B 10.1197004,C -74.1667023,S 2,T 11}
DECL FDAT Fxp12={TOOL_NO 4,BASE_NO 3,IPO_FRAME #BASE,POINT2[] " "}
DECL PDAT PP_OLP14={VEL 100.0,ACC 100.0,APO_DIST 0.0}
DECL E6POS Xxp12={X -2671.84912,Y 1793.97302,Z 566.737,A -2.42820001,B 58.0560989,C 1.01139998,S 2,T 3}
DECL BASIS_SUGG_T LAST_BASIS={POINT1[] "P0                      ",POINT2[] "P0                      ",CP_PARAMS[] "CPDAT0                  ",PTP_PARAMS[] "PDAT0                   ",CONT[] "                        ",CP_VEL[] "2                       ",PTP_VEL[] "100                     ",SPL_NAME[] "S0                      "}
DECL SPOT_SUGG_T LAST_SPOT={GUN[] "2                       ",RETR_CMD[] "#OPN                    ",CHOISE[] "#FIRST                  ",CLO_TM[] "1                       ",PGNO1[] "184                     ",PRESS1[] "0                       ",PGNO2[] "1                       ",PRESS2[] "0                       ",SPOT_PARAMS[] "NORMAL                  "}
DECL E6POS XP1={X -2671.84692,Y 1793.95398,Z 566.742676,A -2.42867708,B 58.05616,C 1.00979102,S 18,T 3,E1 0.0,E2 0.0,E3 0.0,E4 0.0,E5 0.0,E6 0.0}
DECL FDAT FP1={TOOL_NO 4,BASE_NO 3,IPO_FRAME #BASE,POINT2[] " ",TQ_STATE FALSE}
DECL PDAT PPDAT1={VEL 100.0,ACC 100.0,APO_DIST 100.0,GEAR_JERK 50.0}
DECL E6POS XP2={X -1308.08203,Y 274.604095,Z 1383.28406,A -11.6709099,B 10.1234999,C -74.1528397,S 18,T 11,E1 0.0,E2 0.0,E3 0.0,E4 0.0,E5 0.0,E6 0.0}
DECL FDAT FP2={TOOL_NO 4,BASE_NO 3,IPO_FRAME #BASE,POINT2[] " ",TQ_STATE FALSE}
DECL PDAT PPDAT2={VEL 100.0,ACC 100.0,APO_DIST 0.0,APO_MODE #CPTP,GEAR_JERK 50.0}
DECL E6POS XP3={X 178.130798,Y 17.4218903,Z 1098.01904,A 11.9711504,B 9.40271664,C -82.945137,S 18,T 11,E1 0.0,E2 0.0,E3 0.0,E4 0.0,E5 0.0,E6 0.0}
DECL FDAT FP3={TOOL_NO 4,BASE_NO 3,IPO_FRAME #BASE,POINT2[] " ",TQ_STATE FALSE}
DECL PDAT PPDAT3={VEL 100.0,ACC 100.0,APO_DIST 100.0,APO_MODE #CPTP,GEAR_JERK 50.0}
DECL E6POS XP4={X 312.22821,Y 894.042725,Z 1261.80396,A 31.1553802,B -35.6419411,C -56.8302002,S 18,T 11,E1 0.0,E2 0.0,E3 0.0,E4 0.0,E5 0.0,E6 0.0}
DECL FDAT FP4={TOOL_NO 4,BASE_NO 3,IPO_FRAME #BASE,POINT2[] " ",TQ_STATE FALSE}
DECL LDAT LCPDAT1={VEL 2.0,ACC 100.0,APO_DIST 100.0,APO_FAC 50.0,AXIS_VEL 100.0,AXIS_ACC 100.0,ORI_TYP #VAR,CIRC_TYP #BASE,JERK_FAC 50.0,GEAR_JERK 50.0,EXAX_IGN 0}
DECL E6POS XP5={X 363.082703,Y 949.189697,Z 1322.50305,A 36.97995,B -33.8394508,C -64.4538498,S 18,T 11,E1 0.0,E2 0.0,E3 0.0,E4 0.0,E5 0.0,E6 0.0}
DECL FDAT FP5={TOOL_NO 4,BASE_NO 3,IPO_FRAME #BASE,POINT2[] " ",TQ_STATE FALSE}
DECL LDAT LCPDAT2={VEL 2.0,ACC 100.0,APO_DIST 100.0,APO_FAC 50.0,AXIS_VEL 100.0,AXIS_ACC 100.0,ORI_TYP #VAR,CIRC_TYP #BASE,JERK_FAC 50.0,GEAR_JERK 50.0,EXAX_IGN 0}
DECL E6POS XPS01010002={X 363.082489,Y 949.189209,Z 1322.50403,A 36.9799309,B -33.8394585,C -64.4538574,S 18,T 11,E1 0.0,E2 0.0,E3 0.0,E4 0.0,E5 0.0,E6 0.0}
DECL FDAT FPS01010002={TOOL_NO 4,BASE_NO 3,IPO_FRAME #BASE,POINT2[] " ",TQ_STATE FALSE}
DECL PDAT PPDAT4={VEL 100.0,ACC 100.0,APO_DIST 100.0,GEAR_JERK 50.0}
DECL PDAT PP_OLP15={VEL 100.0,ACC 100.0,APO_DIST 0.0}
DECL E6POS XP0={X -1057.83704,Y 966.953003,Z 997.169983,A -179.672302,B -1.48539996,C 179.896301,S 6,T 19}
DECL FDAT FP0={TOOL_NO 5,BASE_NO 0,IPO_FRAME #BASE,POINT2[] " "}
DECL E6POS XP6={X 357.832794,Y 899.258911,Z 1276.77295,A 36.9782715,B -33.8794899,C -62.1634293,S 18,T 11,E1 0.0,E2 0.0,E3 0.0,E4 0.0,E5 0.0,E6 0.0}
DECL FDAT FP6={TOOL_NO 4,BASE_NO 3,IPO_FRAME #BASE,POINT2[] " ",TQ_STATE FALSE}
DECL PDAT PPDAT5={VEL 100.0,ACC 100.0,APO_DIST 100.0,GEAR_JERK 50.0}
DECL E6POS XP7={X 263.495392,Y 575.442505,Z 1201.91101,A 23.1707191,B -19.4270992,C -64.3323898,S 18,T 11,E1 0.0,E2 0.0,E3 0.0,E4 0.0,E5 0.0,E6 0.0}
DECL FDAT FP7={TOOL_NO 4,BASE_NO 3,IPO_FRAME #BASE,POINT2[] " ",TQ_STATE FALSE}
DECL PDAT PPDAT6={VEL 100.0,ACC 100.0,APO_DIST 100.0,APO_MODE #CPTP,GEAR_JERK 50.0}
DECL E6POS XP8={X 312.235413,Y 894.027222,Z 1261.79602,A 31.1545601,B -35.6413383,C -56.8305702,S 18,T 11,E1 0.0,E2 0.0,E3 0.0,E4 0.0,E5 0.0,E6 0.0}
DECL FDAT FP8={TOOL_NO 4,BASE_NO 3,IPO_FRAME #BASE,POINT2[] " ",TQ_STATE FALSE}
DECL PDAT PPDAT7={VEL 100.0,ACC 100.0,APO_DIST 100.0,GEAR_JERK 50.0}
DECL E6POS XP9={X 356.468689,Y 927.755615,Z 1313.48999,A 41.4177094,B -36.3712616,C -63.1682396,S 18,T 11,E1 0.0,E2 0.0,E3 0.0,E4 0.0,E5 0.0,E6 0.0}
DECL FDAT FP9={TOOL_NO 4,BASE_NO 3,IPO_FRAME #BASE,POINT2[] " ",TQ_STATE FALSE}
DECL PDAT PPDAT8={VEL 100.0,ACC 100.0,APO_DIST 100.0,GEAR_JERK 50.0}
DECL E6POS XPS01010003={X 347.886688,Y 915.326599,Z 1325.82397,A 51.0201683,B -39.133419,C -64.2345963,S 18,T 11,E1 0.0,E2 0.0,E3 0.0,E4 0.0,E5 0.0,E6 0.0}
DECL FDAT FPS01010003={TOOL_NO 4,BASE_NO 3,IPO_FRAME #BASE,POINT2[] " ",TQ_STATE FALSE}
DECL PDAT PPDAT9={VEL 100.0,ACC 100.0,APO_DIST 100.0,GEAR_JERK 50.0}
DECL E6POS XP10={X 342.349396,Y 886.705017,Z 1322.31799,A 56.9407005,B -41.1276207,C -62.9248199,S 18,T 11,E1 0.0,E2 0.0,E3 0.0,E4 0.0,E5 0.0,E6 0.0}
DECL FDAT FP10={TOOL_NO 4,BASE_NO 3,IPO_FRAME #BASE,POINT2[] " ",TQ_STATE FALSE}
DECL LDAT LCPDAT3={VEL 2.0,ACC 100.0,APO_DIST 100.0,APO_FAC 50.0,AXIS_VEL 100.0,AXIS_ACC 100.0,ORI_TYP #VAR,CIRC_TYP #BASE,JERK_FAC 50.0,GEAR_JERK 50.0,EXAX_IGN 0}
DECL LDAT LCPDAT4={VEL 2.0,ACC 100.0,APO_DIST 100.0,APO_FAC 50.0,AXIS_VEL 100.0,AXIS_ACC 100.0,ORI_TYP #VAR,CIRC_TYP #BASE,JERK_FAC 50.0,GEAR_JERK 50.0,EXAX_IGN 0}
DECL LDAT LCPDAT5={VEL 2.0,ACC 100.0,APO_DIST 100.0,APO_FAC 50.0,AXIS_VEL 100.0,AXIS_ACC 100.0,ORI_TYP #VAR,CIRC_TYP #BASE,JERK_FAC 50.0,GEAR_JERK 50.0,EXAX_IGN 0}
DECL LDAT LCPDAT6={VEL 2.0,ACC 100.0,APO_DIST 100.0,APO_FAC 50.0,AXIS_VEL 100.0,AXIS_ACC 100.0,ORI_TYP #VAR,CIRC_TYP #BASE,JERK_FAC 50.0,GEAR_JERK 50.0,EXAX_IGN 0}
DECL E6POS XPS01010004={X 333.757599,Y 868.145081,Z 1328.43298,A 56.9288101,B -41.144619,C -62.9054298,S 18,T 11,E1 0.0,E2 0.0,E3 0.0,E4 0.0,E5 0.0,E6 0.0}
DECL FDAT FPS01010004={TOOL_NO 4,BASE_NO 3,IPO_FRAME #BASE,POINT2[] " ",TQ_STATE FALSE}
DECL LDAT LCPDAT7={VEL 2.0,ACC 100.0,APO_DIST 100.0,APO_FAC 50.0,AXIS_VEL 100.0,AXIS_ACC 100.0,ORI_TYP #VAR,CIRC_TYP #BASE,JERK_FAC 50.0,GEAR_JERK 50.0,EXAX_IGN 0}
DECL E6POS XPS01010005={X 326.634399,Y 838.837402,Z 1328.48706,A 64.009613,B -37.8111,C -65.0115967,S 18,T 11,E1 0.0,E2 0.0,E3 0.0,E4 0.0,E5 0.0,E6 0.0}
DECL FDAT FPS01010005={TOOL_NO 4,BASE_NO 3,IPO_FRAME #BASE,POINT2[] " ",TQ_STATE FALSE}
DECL LDAT LCPDAT8={VEL 2.0,ACC 100.0,APO_DIST 100.0,APO_FAC 50.0,AXIS_VEL 100.0,AXIS_ACC 100.0,ORI_TYP #VAR,CIRC_TYP #BASE,JERK_FAC 50.0,GEAR_JERK 50.0,EXAX_IGN 0}
DECL E6POS XPS01010006={X 318.911804,Y 799.581421,Z 1329.73206,A 63.005909,B -41.4448586,C -63.5359993,S 18,T 11,E1 0.0,E2 0.0,E3 0.0,E4 0.0,E5 0.0,E6 0.0}
DECL FDAT FPS01010006={TOOL_NO 4,BASE_NO 3,IPO_FRAME #BASE,POINT2[] " ",TQ_STATE FALSE}
DECL LDAT LCPDAT9={VEL 2.0,ACC 100.0,APO_DIST 100.0,APO_FAC 50.0,AXIS_VEL 100.0,AXIS_ACC 100.0,ORI_TYP #VAR,CIRC_TYP #BASE,JERK_FAC 50.0,GEAR_JERK 50.0,EXAX_IGN 0}
DECL E6POS XPS01010007={X 286.908997,Y -5.12063885,Z 1340.87097,A -81.5047073,B -23.1105499,C 68.9762115,S 18,T 11,E1 0.0,E2 0.0,E3 0.0,E4 0.0,E5 0.0,E6 0.0}
DECL FDAT FPS01010007={TOOL_NO 4,BASE_NO 3,IPO_FRAME #BASE,POINT2[] " ",TQ_STATE FALSE}
DECL LDAT LCPDAT10={VEL 2.0,ACC 100.0,APO_DIST 100.0,APO_FAC 50.0,AXIS_VEL 100.0,AXIS_ACC 100.0,ORI_TYP #VAR,CIRC_TYP #BASE,JERK_FAC 50.0,GEAR_JERK 50.0,EXAX_IGN 0}
DECL E6POS XPS01010008={X 313.420593,Y 758.953186,Z 1332.255,A 65.8980637,B -39.6680107,C -64.0724869,S 18,T 11,E1 0.0,E2 0.0,E3 0.0,E4 0.0,E5 0.0,E6 0.0}
DECL FDAT FPS01010008={TOOL_NO 4,BASE_NO 3,IPO_FRAME #BASE,POINT2[] " ",TQ_STATE FALSE}
DECL LDAT LCPDAT11={VEL 2.0,ACC 100.0,APO_DIST 100.0,APO_FAC 50.0,AXIS_VEL 100.0,AXIS_ACC 100.0,ORI_TYP #VAR,CIRC_TYP #BASE,JERK_FAC 50.0,GEAR_JERK 50.0,EXAX_IGN 0}
DECL E6POS XPS01010009={X 310.396393,Y 721.101196,Z 1331.51794,A 69.3403702,B -38.6280403,C -68.3828735,S 18,T 11,E1 0.0,E2 0.0,E3 0.0,E4 0.0,E5 0.0,E6 0.0}
DECL FDAT FPS01010009={TOOL_NO 4,BASE_NO 3,IPO_FRAME #BASE,POINT2[] " ",TQ_STATE FALSE}
DECL LDAT LCPDAT12={VEL 2.0,ACC 100.0,APO_DIST 100.0,APO_FAC 50.0,AXIS_VEL 100.0,AXIS_ACC 100.0,ORI_TYP #VAR,CIRC_TYP #BASE,JERK_FAC 50.0,GEAR_JERK 50.0,EXAX_IGN 0}
DECL E6POS XP11={X 300.977112,Y 715.575989,Z 1297.76599,A 69.3420563,B -38.630619,C -68.376297,S 18,T 11,E1 0.0,E2 0.0,E3 0.0,E4 0.0,E5 0.0,E6 0.0}
DECL FDAT FP11={TOOL_NO 4,BASE_NO 3,IPO_FRAME #BASE,POINT2[] " ",TQ_STATE FALSE}
DECL LDAT LCPDAT13={VEL 2.0,ACC 100.0,APO_DIST 100.0,APO_FAC 50.0,AXIS_VEL 100.0,AXIS_ACC 100.0,ORI_TYP #VAR,CIRC_TYP #BASE,JERK_FAC 50.0,GEAR_JERK 50.0,EXAX_IGN 0}
DECL E6POS XP12={X 296.070313,Y 611.038574,Z 1292.75,A 70.5039825,B -35.8779716,C -65.223587,S 18,T 11,E1 0.0,E2 0.0,E3 0.0,E4 0.0,E5 0.0,E6 0.0}
DECL FDAT FP12={TOOL_NO 4,BASE_NO 3,IPO_FRAME #BASE,POINT2[] " ",TQ_STATE FALSE}
DECL PDAT PPDAT10={VEL 100.0,ACC 100.0,APO_DIST 100.0,GEAR_JERK 50.0}
DECL LDAT LCPDAT14={VEL 2.0,ACC 100.0,APO_DIST 100.0,APO_FAC 50.0,AXIS_VEL 100.0,AXIS_ACC 100.0,ORI_TYP #VAR,CIRC_TYP #BASE,JERK_FAC 50.0,GEAR_JERK 50.0,EXAX_IGN 0}
DECL E6POS XPS01010010={X 302.343201,Y 618.479187,Z 1332.49304,A 70.4979401,B -35.8856506,C -65.2090073,S 18,T 11,E1 0.0,E2 0.0,E3 0.0,E4 0.0,E5 0.0,E6 0.0}
DECL FDAT FPS01010010={TOOL_NO 4,BASE_NO 3,IPO_FRAME #BASE,POINT2[] " ",TQ_STATE FALSE}
DECL LDAT LCPDAT15={VEL 2.0,ACC 100.0,APO_DIST 100.0,APO_FAC 50.0,AXIS_VEL 100.0,AXIS_ACC 100.0,ORI_TYP #VAR,CIRC_TYP #BASE,JERK_FAC 50.0,GEAR_JERK 50.0,EXAX_IGN 0}
DECL E6POS XP13={X 306.735901,Y 656.108887,Z 1331.59998,A 70.0454788,B -36.9864006,C -66.4973526,S 18,T 11,E1 0.0,E2 0.0,E3 0.0,E4 0.0,E5 0.0,E6 0.0}
DECL FDAT FP13={TOOL_NO 4,BASE_NO 3,IPO_FRAME #BASE,POINT2[] " ",TQ_STATE FALSE}
DECL LDAT LCPDAT16={VEL 2.0,ACC 100.0,APO_DIST 100.0,APO_FAC 50.0,AXIS_VEL 100.0,AXIS_ACC 100.0,ORI_TYP #VAR,CIRC_TYP #BASE,JERK_FAC 50.0,GEAR_JERK 50.0,EXAX_IGN 0}
DECL E6POS XPS01010011={X 298.232208,Y 584.7547,Z 1333.77405,A 71.1074295,B -36.1012993,C -65.1560974,S 18,T 11,E1 0.0,E2 0.0,E3 0.0,E4 0.0,E5 0.0,E6 0.0}
DECL FDAT FPS01010011={TOOL_NO 4,BASE_NO 3,IPO_FRAME #BASE,POINT2[] " ",TQ_STATE FALSE}
DECL LDAT LCPDAT17={VEL 2.0,ACC 100.0,APO_DIST 100.0,APO_FAC 50.0,AXIS_VEL 100.0,AXIS_ACC 100.0,ORI_TYP #VAR,CIRC_TYP #BASE,JERK_FAC 50.0,GEAR_JERK 50.0,EXAX_IGN 0}
DECL E6POS XPS01010012={X 294.127014,Y 478.862915,Z 1336.25098,A 69.2130127,B -41.1254807,C -63.2432289,S 18,T 11,E1 0.0,E2 0.0,E3 0.0,E4 0.0,E5 0.0,E6 0.0}
DECL FDAT FPS01010012={TOOL_NO 4,BASE_NO 3,IPO_FRAME #BASE,POINT2[] " ",TQ_STATE FALSE}
DECL LDAT LCPDAT18={VEL 2.0,ACC 100.0,APO_DIST 100.0,APO_FAC 50.0,AXIS_VEL 100.0,AXIS_ACC 100.0,ORI_TYP #VAR,CIRC_TYP #BASE,JERK_FAC 50.0,GEAR_JERK 50.0,EXAX_IGN 0}
DECL E6POS XP14={X 287.157898,Y 494.053406,Z 1300.08899,A 70.7484131,B -38.73946,C -64.2102966,S 18,T 11,E1 0.0,E2 0.0,E3 0.0,E4 0.0,E5 0.0,E6 0.0}
DECL FDAT FP14={TOOL_NO 4,BASE_NO 3,IPO_FRAME #BASE,POINT2[] " ",TQ_STATE FALSE}
DECL LDAT LCPDAT19={VEL 2.0,ACC 100.0,APO_DIST 100.0,APO_FAC 50.0,AXIS_VEL 100.0,AXIS_ACC 100.0,ORI_TYP #VAR,CIRC_TYP #BASE,JERK_FAC 50.0,GEAR_JERK 50.0,EXAX_IGN 0}
DECL E6POS XP15={X -45.6137886,Y 513.487671,Z 1409.32397,A 70.8332977,B -38.6543503,C -64.2192764,S 18,T 11,E1 0.0,E2 0.0,E3 0.0,E4 0.0,E5 0.0,E6 0.0}
DECL FDAT FP15={TOOL_NO 4,BASE_NO 3,IPO_FRAME #BASE,POINT2[] " ",TQ_STATE FALSE}
DECL PDAT PPDAT11={VEL 100.0,ACC 100.0,APO_DIST 100.0,GEAR_JERK 50.0}
DECL E6POS XP16={X -45.64468,Y 513.591309,Z 1409.22998,A 70.8363876,B -38.6498413,C -64.2175827,S 18,T 11,E1 0.0,E2 0.0,E3 0.0,E4 0.0,E5 0.0,E6 0.0}
DECL FDAT FP16={TOOL_NO 4,BASE_NO 3,IPO_FRAME #BASE,POINT2[] " ",TQ_STATE FALSE}
DECL PDAT PPDAT12={VEL 100.0,ACC 100.0,APO_DIST 100.0,GEAR_JERK 50.0}
DECL E6POS XP17={X -18.0078106,Y 226.764603,Z 1528.60999,A -52.235611,B -66.3029099,C 40.4377289,S 18,T 11,E1 0.0,E2 0.0,E3 0.0,E4 0.0,E5 0.0,E6 0.0}
DECL FDAT FP17={TOOL_NO 4,BASE_NO 3,IPO_FRAME #BASE,POINT2[] " ",TQ_STATE FALSE}
DECL PDAT PPDAT13={VEL 100.0,ACC 100.0,APO_DIST 0.0,APO_MODE #CPTP,GEAR_JERK 50.0}
DECL PDAT PP_OLP16={VEL 100.0,ACC 100.0,APO_DIST 0.0}
DECL E6POS XP18={X -1057.83704,Y 966.953003,Z 997.169983,A -179.672302,B -1.48539996,C 179.896301,S 6,T 19}
DECL FDAT FP18={TOOL_NO 5,BASE_NO 0,IPO_FRAME #BASE,POINT2[] " "}
DECL E6POS XP19={X -577.50647,Y 1201.73401,Z 2360.15405,A 118.668198,B -28.3075809,C -41.1689491,S 18,T 11,E1 0.0,E2 0.0,E3 0.0,E4 0.0,E5 0.0,E6 0.0}
DECL FDAT FP19={TOOL_NO 5,BASE_NO 0,IPO_FRAME #BASE,POINT2[] " ",TQ_STATE FALSE}
DECL PDAT PPDAT14={VEL 100.0,ACC 100.0,APO_DIST 0.0,APO_MODE #CPTP,GEAR_JERK 50.0}
DECL E6POS XP20={X -820.111572,Y 1456.91602,Z 2354.62207,A 113.311401,B -15.3934002,C -27.9882107,S 18,T 11,E1 0.0,E2 0.0,E3 0.0,E4 0.0,E5 0.0,E6 0.0}
DECL FDAT FP20={TOOL_NO 5,BASE_NO 0,IPO_FRAME #BASE,POINT2[] " ",TQ_STATE FALSE}
DECL PDAT PPDAT15={VEL 100.0,ACC 100.0,APO_DIST 100.0,GEAR_JERK 50.0}
DECL E6POS XPS01010013={X 287.224915,Y 46.7158699,Z 1340.98499,A -82.1270294,B -22.1040993,C 69.1398621,S 18,T 11,E1 0.0,E2 0.0,E3 0.0,E4 0.0,E5 0.0,E6 0.0}
DECL FDAT FPS01010013={TOOL_NO 4,BASE_NO 3,IPO_FRAME #BASE,POINT2[] " ",TQ_STATE FALSE}
DECL LDAT LCPDAT20={VEL 2.0,ACC 100.0,APO_DIST 100.0,APO_FAC 50.0,AXIS_VEL 100.0,AXIS_ACC 100.0,ORI_TYP #VAR,CIRC_TYP #BASE,JERK_FAC 50.0,GEAR_JERK 50.0,EXAX_IGN 0}
DECL E6POS XPS01010014={X 287.073303,Y -54.0063591,Z 1341.10303,A -81.0786972,B -23.4212208,C 68.9073334,S 18,T 11,E1 0.0,E2 0.0,E3 0.0,E4 0.0,E5 0.0,E6 0.0}
DECL FDAT FPS01010014={TOOL_NO 4,BASE_NO 3,IPO_FRAME #BASE,POINT2[] " ",TQ_STATE FALSE}
DECL LDAT LCPDAT21={VEL 2.0,ACC 100.0,APO_DIST 100.0,APO_FAC 50.0,AXIS_VEL 100.0,AXIS_ACC 100.0,ORI_TYP #VAR,CIRC_TYP #BASE,JERK_FAC 50.0,GEAR_JERK 50.0,EXAX_IGN 0}
DECL E6POS XPS01010015={X 287.761414,Y -158.061493,Z 1340.63196,A -81.3838882,B -21.8413296,C 69.1773529,S 18,T 11,E1 0.0,E2 0.0,E3 0.0,E4 0.0,E5 0.0,E6 0.0}
DECL FDAT FPS01010015={TOOL_NO 4,BASE_NO 3,IPO_FRAME #BASE,POINT2[] " ",TQ_STATE FALSE}
DECL LDAT LCPDAT22={VEL 2.0,ACC 100.0,APO_DIST 100.0,APO_FAC 50.0,AXIS_VEL 100.0,AXIS_ACC 100.0,ORI_TYP #VAR,CIRC_TYP #BASE,JERK_FAC 50.0,GEAR_JERK 50.0,EXAX_IGN 0}
DECL E6POS XPS01010016={X 287.738312,Y -208.118607,Z 1339.63599,A -81.4336777,B -21.0888004,C 69.494133,S 18,T 11,E1 0.0,E2 0.0,E3 0.0,E4 0.0,E5 0.0,E6 0.0}
DECL FDAT FPS01010016={TOOL_NO 4,BASE_NO 3,IPO_FRAME #BASE,POINT2[] " ",TQ_STATE FALSE}
DECL LDAT LCPDAT23={VEL 2.0,ACC 100.0,APO_DIST 100.0,APO_FAC 50.0,AXIS_VEL 100.0,AXIS_ACC 100.0,ORI_TYP #VAR,CIRC_TYP #BASE,JERK_FAC 50.0,GEAR_JERK 50.0,EXAX_IGN 0}
DECL E6POS XPS01010017={X 289.020386,Y -261.987091,Z 1338.72998,A -80.2098312,B -22.9787693,C 69.1293335,S 18,T 11,E1 0.0,E2 0.0,E3 0.0,E4 0.0,E5 0.0,E6 0.0}
DECL FDAT FPS01010017={TOOL_NO 4,BASE_NO 3,IPO_FRAME #BASE,POINT2[] " ",TQ_STATE FALSE}
DECL LDAT LCPDAT24={VEL 2.0,ACC 100.0,APO_DIST 100.0,APO_FAC 50.0,AXIS_VEL 100.0,AXIS_ACC 100.0,ORI_TYP #VAR,CIRC_TYP #BASE,JERK_FAC 50.0,GEAR_JERK 50.0,EXAX_IGN 0}
DECL E6POS XPS01010018={X 289.928314,Y -314.829407,Z 1338.43799,A -80.3265686,B -22.3762207,C 69.0457535,S 18,T 11,E1 0.0,E2 0.0,E3 0.0,E4 0.0,E5 0.0,E6 0.0}
DECL FDAT FPS01010018={TOOL_NO 4,BASE_NO 3,IPO_FRAME #BASE,POINT2[] " ",TQ_STATE FALSE}
DECL LDAT LCPDAT25={VEL 2.0,ACC 100.0,APO_DIST 100.0,APO_FAC 50.0,AXIS_VEL 100.0,AXIS_ACC 100.0,ORI_TYP #VAR,CIRC_TYP #BASE,JERK_FAC 50.0,GEAR_JERK 50.0,EXAX_IGN 0}
DECL E6POS XPS01010019={X 291.444794,Y -365.881714,Z 1338.10205,A -80.1103134,B -22.1441898,C 69.3087463,S 18,T 11,E1 0.0,E2 0.0,E3 0.0,E4 0.0,E5 0.0,E6 0.0}
DECL FDAT FPS01010019={TOOL_NO 4,BASE_NO 3,IPO_FRAME #BASE,POINT2[] " ",TQ_STATE FALSE}
DECL LDAT LCPDAT26={VEL 2.0,ACC 100.0,APO_DIST 100.0,APO_FAC 50.0,AXIS_VEL 100.0,AXIS_ACC 100.0,ORI_TYP #VAR,CIRC_TYP #BASE,JERK_FAC 50.0,GEAR_JERK 50.0,EXAX_IGN 0}
DECL E6POS XPS01010020={X 295.380096,Y -472.567413,Z 1336.38696,A -79.1937866,B -22.2749691,C 68.9143982,S 18,T 11,E1 0.0,E2 0.0,E3 0.0,E4 0.0,E5 0.0,E6 0.0}
DECL FDAT FPS01010020={TOOL_NO 4,BASE_NO 3,IPO_FRAME #BASE,POINT2[] " ",TQ_STATE FALSE}
DECL LDAT LCPDAT27={VEL 2.0,ACC 100.0,APO_DIST 100.0,APO_FAC 50.0,AXIS_VEL 100.0,AXIS_ACC 100.0,ORI_TYP #VAR,CIRC_TYP #BASE,JERK_FAC 50.0,GEAR_JERK 50.0,EXAX_IGN 0}
DECL E6POS XPS01010021={X 297.546814,Y -524.037476,Z 1335.75806,A -79.584938,B -20.0944901,C 69.1831894,S 18,T 11,E1 0.0,E2 0.0,E3 0.0,E4 0.0,E5 0.0,E6 0.0}
DECL FDAT FPS01010021={TOOL_NO 4,BASE_NO 3,IPO_FRAME #BASE,POINT2[] " ",TQ_STATE FALSE}
DECL LDAT LCPDAT28={VEL 2.0,ACC 100.0,APO_DIST 100.0,APO_FAC 50.0,AXIS_VEL 100.0,AXIS_ACC 100.0,ORI_TYP #VAR,CIRC_TYP #BASE,JERK_FAC 50.0,GEAR_JERK 50.0,EXAX_IGN 0}
DECL PDAT PP_OLP17={VEL 100.0,ACC 100.0,APO_DIST 0.0}
DECL E6POS XP21={X -1057.83704,Y 966.953003,Z 997.169983,A -179.672302,B -1.48539996,C 179.896301,S 6,T 19}
DECL FDAT FP21={TOOL_NO 5,BASE_NO 0,IPO_FRAME #BASE,POINT2[] " "}
DECL E6POS XPS01010022={X 303.966614,Y -620.996887,Z 1331.75098,A -78.1263733,B -20.25214,C 69.1010895,S 18,T 11,E1 0.0,E2 0.0,E3 0.0,E4 0.0,E5 0.0,E6 0.0}
DECL FDAT FPS01010022={TOOL_NO 4,BASE_NO 3,IPO_FRAME #BASE,POINT2[] " ",TQ_STATE FALSE}
DECL LDAT LCPDAT29={VEL 2.0,ACC 100.0,APO_DIST 100.0,APO_FAC 50.0,AXIS_VEL 100.0,AXIS_ACC 100.0,ORI_TYP #VAR,CIRC_TYP #BASE,JERK_FAC 50.0,GEAR_JERK 50.0,EXAX_IGN 0}
DECL E6POS XPS01010023={X 311.523102,Y -720.246826,Z 1331.91699,A -76.8176804,B -20.4881496,C 68.9858322,S 18,T 11,E1 0.0,E2 0.0,E3 0.0,E4 0.0,E5 0.0,E6 0.0}
DECL FDAT FPS01010023={TOOL_NO 4,BASE_NO 3,IPO_FRAME #BASE,POINT2[] " ",TQ_STATE FALSE}
DECL LDAT LCPDAT30={VEL 2.0,ACC 100.0,APO_DIST 100.0,APO_FAC 50.0,AXIS_VEL 100.0,AXIS_ACC 100.0,ORI_TYP #VAR,CIRC_TYP #BASE,JERK_FAC 50.0,GEAR_JERK 50.0,EXAX_IGN 0}
DECL E6POS XPS01010024={X 315.40741,Y -759.460388,Z 1330.33398,A -76.547493,B -18.2475204,C 69.2206802,S 18,T 11,E1 0.0,E2 0.0,E3 0.0,E4 0.0,E5 0.0,E6 0.0}
DECL FDAT FPS01010024={TOOL_NO 4,BASE_NO 3,IPO_FRAME #BASE,POINT2[] " ",TQ_STATE FALSE}
DECL LDAT LCPDAT31={VEL 2.0,ACC 100.0,APO_DIST 100.0,APO_FAC 50.0,AXIS_VEL 100.0,AXIS_ACC 100.0,ORI_TYP #VAR,CIRC_TYP #BASE,JERK_FAC 50.0,GEAR_JERK 50.0,EXAX_IGN 0}
DECL E6POS XPS01010025={X 320.685211,Y -798.215576,Z 1329.48804,A -74.3228836,B -18.2347298,C 69.5574722,S 18,T 11,E1 0.0,E2 0.0,E3 0.0,E4 0.0,E5 0.0,E6 0.0}
DECL FDAT FPS01010025={TOOL_NO 4,BASE_NO 3,IPO_FRAME #BASE,POINT2[] " ",TQ_STATE FALSE}
DECL LDAT LCPDAT32={VEL 2.0,ACC 100.0,APO_DIST 100.0,APO_FAC 50.0,AXIS_VEL 100.0,AXIS_ACC 100.0,ORI_TYP #VAR,CIRC_TYP #BASE,JERK_FAC 50.0,GEAR_JERK 50.0,EXAX_IGN 0}
DECL E6POS XPS01010026={X 326.906586,Y -835.311218,Z 1328.21899,A -72.3317108,B -19.9759293,C 69.1068573,S 18,T 11,E1 0.0,E2 0.0,E3 0.0,E4 0.0,E5 0.0,E6 0.0}
DECL FDAT FPS01010026={TOOL_NO 4,BASE_NO 3,IPO_FRAME #BASE,POINT2[] " ",TQ_STATE FALSE}
DECL LDAT LCPDAT33={VEL 2.0,ACC 100.0,APO_DIST 100.0,APO_FAC 50.0,AXIS_VEL 100.0,AXIS_ACC 100.0,ORI_TYP #VAR,CIRC_TYP #BASE,JERK_FAC 50.0,GEAR_JERK 50.0,EXAX_IGN 0}
DECL E6POS XPS01010027={X 334.537292,Y -868.387512,Z 1324.54504,A -72.3300629,B -19.9233608,C 69.1167221,S 18,T 11,E1 0.0,E2 0.0,E3 0.0,E4 0.0,E5 0.0,E6 0.0}
DECL FDAT FPS01010027={TOOL_NO 4,BASE_NO 3,IPO_FRAME #BASE,POINT2[] " ",TQ_STATE FALSE}
DECL LDAT LCPDAT34={VEL 2.0,ACC 100.0,APO_DIST 100.0,APO_FAC 50.0,AXIS_VEL 100.0,AXIS_ACC 100.0,ORI_TYP #VAR,CIRC_TYP #BASE,JERK_FAC 50.0,GEAR_JERK 50.0,EXAX_IGN 0}
DECL E6POS XP22={X 350.80069,Y -907.980713,Z 1321.32397,A -60.67313,B -19.5815105,C 69.0403671,S 18,T 11,E1 0.0,E2 0.0,E3 0.0,E4 0.0,E5 0.0,E6 0.0}
DECL FDAT FP22={TOOL_NO 4,BASE_NO 3,IPO_FRAME #BASE,POINT2[] " ",TQ_STATE FALSE}
DECL LDAT LCPDAT35={VEL 2.0,ACC 100.0,APO_DIST 100.0,APO_FAC 50.0,AXIS_VEL 100.0,AXIS_ACC 100.0,ORI_TYP #VAR,CIRC_TYP #BASE,JERK_FAC 50.0,GEAR_JERK 50.0,EXAX_IGN 0}
DECL E6POS XPS01010028={X 346.304108,Y -910.412292,Z 1321.62305,A -60.6612892,B -19.5378704,C 69.027977,S 18,T 11,E1 0.0,E2 0.0,E3 0.0,E4 0.0,E5 0.0,E6 0.0}
DECL FDAT FPS01010028={TOOL_NO 4,BASE_NO 3,IPO_FRAME #BASE,POINT2[] " ",TQ_STATE FALSE}
DECL LDAT LCPDAT36={VEL 2.0,ACC 100.0,APO_DIST 100.0,APO_FAC 50.0,AXIS_VEL 100.0,AXIS_ACC 100.0,ORI_TYP #VAR,CIRC_TYP #BASE,JERK_FAC 50.0,GEAR_JERK 50.0,EXAX_IGN 0}
DECL E6POS XP23={X 350.461609,Y -908.779419,Z 1317.86401,A -60.6727715,B -19.5289097,C 69.0452194,S 18,T 11,E1 0.0,E2 0.0,E3 0.0,E4 0.0,E5 0.0,E6 0.0}
DECL FDAT FP23={TOOL_NO 4,BASE_NO 3,IPO_FRAME #BASE,POINT2[] " ",TQ_STATE FALSE}
DECL LDAT LCPDAT37={VEL 2.0,ACC 100.0,APO_DIST 100.0,APO_FAC 50.0,AXIS_VEL 100.0,AXIS_ACC 100.0,ORI_TYP #VAR,CIRC_TYP #BASE,JERK_FAC 50.0,GEAR_JERK 50.0,EXAX_IGN 0}
DECL E6POS XP24={X 377.234802,Y -954.668274,Z 1303.73999,A -49.9476204,B -14.7396402,C 71.581337,S 18,T 11,E1 0.0,E2 0.0,E3 0.0,E4 0.0,E5 0.0,E6 0.0}
DECL FDAT FP24={TOOL_NO 4,BASE_NO 3,IPO_FRAME #BASE,POINT2[] " ",TQ_STATE FALSE}
DECL LDAT LCPDAT38={VEL 2.0,ACC 100.0,APO_DIST 100.0,APO_FAC 50.0,AXIS_VEL 100.0,AXIS_ACC 100.0,ORI_TYP #VAR,CIRC_TYP #BASE,JERK_FAC 50.0,GEAR_JERK 50.0,EXAX_IGN 0}
DECL E6POS XP25={X 350.251099,Y -972.364075,Z 1294.35999,A -47.8951492,B -6.4500351,C -108.647697,S 18,T 43,E1 0.0,E2 0.0,E3 0.0,E4 0.0,E5 0.0,E6 0.0}
DECL FDAT FP25={TOOL_NO 4,BASE_NO 3,IPO_FRAME #BASE,POINT2[] " ",TQ_STATE FALSE}
DECL LDAT LCPDAT39={VEL 2.0,ACC 100.0,APO_DIST 100.0,APO_FAC 50.0,AXIS_VEL 100.0,AXIS_ACC 100.0,ORI_TYP #VAR,CIRC_TYP #BASE,JERK_FAC 50.0,GEAR_JERK 50.0,EXAX_IGN 0}
DECL E6POS XPS01010029={X 366.317108,Y -956.599609,Z 1312.99097,A -49.9479599,B -14.7375898,C 71.5824585,S 18,T 11,E1 0.0,E2 0.0,E3 0.0,E4 0.0,E5 0.0,E6 0.0}
DECL FDAT FPS01010029={TOOL_NO 4,BASE_NO 3,IPO_FRAME #BASE,POINT2[] " ",TQ_STATE FALSE}
DECL LDAT LCPDAT40={VEL 2.0,ACC 100.0,APO_DIST 100.0,APO_FAC 50.0,AXIS_VEL 100.0,AXIS_ACC 100.0,ORI_TYP #VAR,CIRC_TYP #BASE,JERK_FAC 50.0,GEAR_JERK 50.0,EXAX_IGN 0}
DECL E6POS XP26={X 317.417603,Y -945.340698,Z 1268.61304,A -31.6410809,B 2.5564599,C -115.785202,S 18,T 43,E1 0.0,E2 0.0,E3 0.0,E4 0.0,E5 0.0,E6 0.0}
DECL FDAT FP26={TOOL_NO 4,BASE_NO 3,IPO_FRAME #BASE,POINT2[] " ",TQ_STATE FALSE}
DECL PDAT PPDAT16={VEL 100.0,ACC 100.0,APO_DIST 0.0,APO_MODE #CPTP,GEAR_JERK 50.0}
DECL E6POS XP27={X -58.2851982,Y -984.979187,Z 1087.82703,A -53.9089394,B 30.2852993,C -162.633301,S 18,T 11,E1 0.0,E2 0.0,E3 0.0,E4 0.0,E5 0.0,E6 0.0}
DECL FDAT FP27={TOOL_NO 4,BASE_NO 3,IPO_FRAME #BASE,POINT2[] " ",TQ_STATE FALSE}
DECL PDAT PPDAT17={VEL 100.0,ACC 100.0,APO_DIST 0.0,APO_MODE #CPTP,GEAR_JERK 50.0}
DECL E6POS XP28={X -239.330093,Y -983.23877,Z 1069.04199,A -69.4001465,B 23.2971592,C 148.591293,S 18,T 11,E1 0.0,E2 0.0,E3 0.0,E4 0.0,E5 0.0,E6 0.0}
DECL FDAT FP28={TOOL_NO 4,BASE_NO 3,IPO_FRAME #BASE,POINT2[] " ",TQ_STATE FALSE}
DECL PDAT PPDAT18={VEL 100.0,ACC 100.0,APO_DIST 0.0,APO_MODE #CPTP,GEAR_JERK 50.0}
DECL E6POS XP29={X 358.162415,Y -920.245728,Z 1275.31799,A -49.9455185,B -14.7352505,C 71.5783768,S 18,T 11,E1 0.0,E2 0.0,E3 0.0,E4 0.0,E5 0.0,E6 0.0}
DECL FDAT FP29={TOOL_NO 4,BASE_NO 3,IPO_FRAME #BASE,POINT2[] " ",TQ_STATE FALSE}
DECL LDAT LCPDAT41={VEL 2.0,ACC 100.0,APO_DIST 100.0,APO_FAC 50.0,AXIS_VEL 100.0,AXIS_ACC 100.0,ORI_TYP #VAR,CIRC_TYP #BASE,JERK_FAC 50.0,GEAR_JERK 50.0,EXAX_IGN 0}
DECL E6POS XP30={X 89.4211121,Y -806.234619,Z 1282.526,A -55.1771584,B -14.5796499,C 75.1306763,S 18,T 11,E1 0.0,E2 0.0,E3 0.0,E4 0.0,E5 0.0,E6 0.0}
DECL FDAT FP30={TOOL_NO 4,BASE_NO 3,IPO_FRAME #BASE,POINT2[] " ",TQ_STATE FALSE}
DECL PDAT PPDAT19={VEL 100.0,ACC 100.0,APO_DIST 0.0,APO_MODE #CPTP,GEAR_JERK 50.0}
DECL E6POS XP31={X -1308.07898,Y 274.512787,Z 1383.53198,A -11.6748104,B 10.1168604,C -74.1650467,S 18,T 11,E1 0.0,E2 0.0,E3 0.0,E4 0.0,E5 0.0,E6 0.0}
DECL FDAT FP31={TOOL_NO 4,BASE_NO 3,IPO_FRAME #BASE,POINT2[] " ",TQ_STATE FALSE}
DECL PDAT PPDAT20={VEL 100.0,ACC 50.0,APO_DIST 0.0,APO_MODE #CPTP,GEAR_JERK 50.0}
DECL E6POS XP32={X -2671.823,Y 1793.96204,Z 566.747681,A -2.41564012,B 58.0559502,C 1.00735104,S 18,T 3,E1 0.0,E2 0.0,E3 0.0,E4 0.0,E5 0.0,E6 0.0}
DECL FDAT FP32={TOOL_NO 4,BASE_NO 3,IPO_FRAME #BASE,POINT2[] " ",TQ_STATE FALSE}
DECL PDAT PPDAT21={VEL 100.0,ACC 100.0,APO_DIST 100.0,GEAR_JERK 50.0}
DECL E6POS XP33={X -2671.82593,Y 1793.96106,Z 566.747375,A -2.415416,B 58.0559311,C 1.00737596,S 18,T 3,E1 0.0,E2 0.0,E3 0.0,E4 0.0,E5 0.0,E6 0.0}
DECL FDAT FP33={TOOL_NO 4,BASE_NO 3,IPO_FRAME #BASE,POINT2[] " ",TQ_STATE FALSE}
DECL PDAT PPDAT22={VEL 100.0,ACC 100.0,APO_DIST 100.0,GEAR_JERK 50.0}
ENDDAT
